# B&R Automation Studio project NAELD004C00R10L518F00 (part 37)

#### Act_Background.st
```iecst
(** 2019-01-21 **)
ACTION Act_Background:

	//Digital Input Mapping With Physical Input
	IF p_tyDISettings.diSafetyRlySig > 0 AND p_tyDISettings.diSafetyRlySig <= UDINT_TO_DINT(p_udiMax) THEN
		tyDInput.bSafetyRlySig	:= a_bPhysicalDI[p_tyDISettings.diSafetyRlySig];
	ELSE
		tyDInput.bSafetyRlySig	:= TRUE;
	END_IF

	IF p_tyDISettings.diEStopSig > 0 AND p_tyDISettings.diEStopSig <= UDINT_TO_DINT(p_udiMax) THEN
		tyDInput.bEStopSig	:= a_bPhysicalDI[p_tyDISettings.diEStopSig];
	ELSE
		tyDInput.bEStopSig	:= TRUE;
	END_IF

	IF p_tyDISettings.diCoverSWSig > 0 AND p_tyDISettings.diCoverSWSig <= UDINT_TO_DINT(p_udiMax) THEN
		tyDInput.bCoverSWSig	:= a_bPhysicalDI[p_tyDISettings.diCoverSWSig];
	ELSE
		tyDInput.bCoverSWSig	:= TRUE;
	END_IF

	IF bSelfTest = FALSE THEN
		IF p_tyDISettings.diDSBA > 0 AND p_tyDISettings.diDSBA <= UDINT_TO_DINT(p_udiMax) THEN
			tyDInput.bDSBA	:= a_bPhysicalDI[p_tyDISettings.diDSBA];
		ELSE
			tyDInput.bDSBA	:= FALSE;
		END_IF
	ELSE
		tyDInput.bDSBA	:= p_bPullConvHvBrd;
	END_IF

	IF p_tyDISettings.diDSBB > 0 AND p_tyDISettings.diDSBB <= UDINT_TO_DINT(p_udiMax) THEN
		tyDInput.bDSBB	:= a_bPhysicalDI[p_tyDISettings.diDSBB];
	ELSE
		tyDInput.bDSBB	:= FALSE;
	END_IF

	IF p_tyDISettings.diPullerExtRS > 0 AND p_tyDISettings.diPullerExtRS <= UDINT_TO_DINT(p_udiMax) THEN
		tyDInput.bPullerExtRS	:= a_bPhysicalDI[p_tyDISettings.diPullerExtRS];
	ELSE
		tyDInput.bPullerExtRS	:= FALSE;
	END_IF

	IF p_tyDISettings.diPullerRetRS > 0 AND p_tyDISettings.diPullerRetRS <= UDINT_TO_DINT(p_udiMax) THEN
		tyDInput.bPullerRetRS	:= a_bPhysicalDI[p_tyDISettings.diPullerRetRS];
	ELSE
		tyDInput.bPullerRetRS	:= TRUE;
	END_IF

	IF p_tyDISettings.diPullerRotHmRS > 0 AND p_tyDISettings.diPullerRotHmRS <= UDINT_TO_DINT(p_udiMax) THEN
		tyDInput.bPullerRotHmRS	:= a_bPhysicalDI[p_tyDISettings.diPullerRotHmRS];
	ELSE
		tyDInput.bPullerRotHmRS	:= TRUE;
	END_IF

	IF p_tyDISettings.diPullerRotRmRS > 0 AND p_tyDISettings.diPullerRotRmRS <= UDINT_TO_DINT(p_udiMax) THEN
		tyDInput.bPullerRotRmRS	:= a_bPhysicalDI[p_tyDISettings.diPullerRotRmRS];
	ELSE
		tyDInput.bPullerRotRmRS	:= FALSE;
	END_IF

	IF bSelfTest = FALSE THEN
		IF p_tyDISettings.diConvLftSen > 0 AND p_tyDISettings.diConvLftSen <= UDINT_TO_DINT(p_udiMax) THEN
			//Digital Input Filter
			fbConvLftSigFltr.tSigOnFltrTm	:= DINT_TO_TIME(p_diConvLftSenOnTm);
			fbConvLftSigFltr.tSigOffFltrTm	:= DINT_TO_TIME(p_diConvLftSenOffTm);
			fbConvLftSigFltr(bSigIn := a_bPhysicalDI[p_tyDISettings.diConvLftSen]);

			tyDInput.bConvLftSen	:= fbConvLftSigFltr.bSigOut;
		ELSE
			tyDInput.bConvLftSen	:= FALSE;
		END_IF
	ELSE
//		fbConvLftSenTm(IN:= p_bPullConvHvBrd);
//		IF EDGEPOS(p_bPullConvHvBrd) THEN
//			tyDInput.bConvLftSen	:= TRUE;
//		ELSIF fbConvLftSenTm.Q THEN
//			tyDInput.bConvLftSen	:= FALSE;
//		END_IF
	END_IF

	IF bSelfTest = FALSE THEN
		IF p_tyDISettings.diConvRgtSen > 0 AND p_tyDISettings.diConvRgtSen <= UDINT_TO_DINT(p_udiMax) THEN
			//Digital Input Filter
			fbConvRgtSigFltr.tSigOnFltrTm	:= DINT_TO_TIME(p_diConvRgtSenOnTm);
			fbConvRgtSigFltr.tSigOffFltrTm	:= DINT_TO_TIME(p_diConvRgtSenOffTm);
			fbConvRgtSigFltr(bSigIn := a_bPhysicalDI[p_tyDISettings.diConvRgtSen]);
			tyDInput.bConvRgtSen	:= fbConvRgtSigFltr.bSigOut;
		ELSE
			tyDInput.bConvRgtSen	:= FALSE;
		END_IF
	ELSE
		tyDInput.bConvRgtSen	:= p_bPullConvHvBrd;
	END_IF

	IF p_tyDISettings.diLifterTimingBeltSen > 0 AND p_tyDISettings.diLifterTimingBeltSen <= UDINT_TO_DINT(p_udiMax) THEN
		tyDInput.bLifterTimingBeltSen	:= a_bPhysicalDI[p_tyDISettings.diLifterTimingBeltSen];
	ELSE
		tyDInput.bLifterTimingBeltSen	:= TRUE;
	END_IF

	IF p_tyDISettings.diLifterSafetyLmtSW1 > 0 AND p_tyDISettings.diLifterSafetyLmtSW1 <= UDINT_TO_DINT(p_udiMax) THEN
		tyDInput.bLifterSafetyLmtSW1	:= a_bPhysicalDI[p_tyDISettings.diLifterSafetyLmtSW1];
	ELSE
		tyDInput.bLifterSafetyLmtSW1	:= TRUE;
	END_IF

	IF p_tyDISettings.diLifterSafetyLmtSW2 > 0 AND p_tyDISettings.diLifterSafetyLmtSW2 <= UDINT_TO_DINT(p_udiMax) THEN
		tyDInput.bLifterSafetyLmtSW2	:= a_bPhysicalDI[p_tyDISettings.diLifterSafetyLmtSW2];
	ELSE
		tyDInput.bLifterSafetyLmtSW2	:= TRUE;
	END_IF

	//Magazine 1 Fixed Clamper RSs
	IF p_tyDISettings.diMag1FixedClampRS > 0 AND p_tyDISettings.diMag1FixedClampRS <= UDINT_TO_DINT(p_udiMax) THEN
		tyDInput.bMag1FixedClampRS	:= a_bPhysicalDI[p_tyDISettings.diMag1FixedClampRS];
	ELSE
		tyDInput.bMag1FixedClampRS	:= FALSE;
	END_IF

	IF p_tyDISettings.diMag1FixedUnclampRS > 0 AND p_tyDISettings.diMag1FixedUnclampRS <= UDINT_TO_DINT(p_udiMax) THEN
		tyDInput.bMag1FixedUnclampRS	:= a_bPhysicalDI[p_tyDISettings.diMag1FixedUnclampRS];
	ELSE
		tyDInput.bMag1FixedUnclampRS	:= TRUE;
	END_IF

	//Magazine 1 Remote Clamper RSs
	IF p_tyDISettings.diMag1RemoteClampRS > 0 AND p_tyDISettings.diMag1RemoteClampRS <= UDINT_TO_DINT(p_udiMax) THEN
		tyDInput.bMag1RemoteClampRS	:= a_bPhysicalDI[p_tyDISettings.diMag1RemoteClampRS];
	ELSE
		tyDInput.bMag1RemoteClampRS	:= FALSE;
	END_IF

	IF p_tyDISettings.diMag1RemoteUnclampRS > 0 AND p_tyDISettings.diMag1RemoteUnclampRS <= UDINT_TO_DINT(p_udiMax) THEN
		tyDInput.bMag1RemoteUnclampRS	:= a_bPhysicalDI[p_tyDISettings.diMag1RemoteUnclampRS];
	ELSE
		tyDInput.bMag1RemoteUnclampRS	:= TRUE;
	END_IF

	//Magazine 1 Sel Clamper RSs
	IF p_tyDISettings.diMag1SelUnClampRS > 0 AND p_tyDISettings.diMag1SelUnClampRS <= UDINT_TO_DINT(p_udiMax) THEN
		tyDInput.bMag1SelUnClampRS	:= a_bPhysicalDI[p_tyDISettings.diMag1SelUnClampRS];
	ELSE
		tyDInput.bMag1SelUnClampRS	:= FALSE;
	END_IF

	//Magazine 2 Fixed Clamper RSs
	IF p_tyDISettings.diMag2FixedClampRS > 0 AND p_tyDISettings.diMag2FixedClampRS <= UDINT_TO_DINT(p_udiMax) THEN
		tyDInput.bMag2FixedClampRS	:= a_bPhysicalDI[p_tyDISettings.diMag2FixedClampRS];
	ELSE
		tyDInput.bMag2FixedClampRS	:= FALSE;
	END_IF

	IF p_tyDISettings.diMag2FixedUnclampRS > 0 AND p_tyDISettings.diMag2FixedUnclampRS <= UDINT_TO_DINT(p_udiMax) THEN
		tyDInput.bMag2FixedUnclampRS	:= a_bPhysicalDI[p_tyDISettings.diMag2FixedUnclampRS];
	ELSE
		tyDInput.bMag2FixedUnclampRS	:= TRUE;
	END_IF

	//Magazine 2 Remote Clamper RSs
	IF p_tyDISettings.diMag2RemoteClampRS > 0 AND p_tyDISettings.diMag2RemoteClampRS <= UDINT_TO_DINT(p_udiMax) THEN
		tyDInput.bMag2RemoteClampRS	:= a_bPhysicalDI[p_tyDISettings.diMag2RemoteClampRS];
	ELSE
		tyDInput.bMag2RemoteClampRS	:= FALSE;
	END_IF

	IF p_tyDISettings.diMag2RemoteUnclampRS > 0 AND p_tyDISettings.diMag2RemoteUnclampRS <= UDINT_TO_DINT(p_udiMax) THEN
		tyDInput.bMag2RemoteUnclampRS	:= a_bPhysicalDI[p_tyDISettings.diMag2RemoteUnclampRS];
	ELSE
		tyDInput.bMag2RemoteUnclampRS	:= TRUE;
	END_IF

	//Magazine 2 Sel Clamper RSs
	IF p_tyDISettings.diMag2SelUnClampRS > 0 AND p_tyDISettings.diMag2SelUnClampRS <= UDINT_TO_DINT(p_udiMax) THEN
		tyDInput.bMag2SelUnClampRS	:= a_bPhysicalDI[p_tyDISettings.diMag2SelUnClampRS];
	ELSE
		tyDInput.bMag2SelUnClampRS	:= FALSE;
	END_IF

	//Magazine 3 Fixed Clamper RSs
	IF p_tyDISettings.diMag3FixedClampRS > 0 AND p_tyDISettings.diMag3FixedClampRS <= UDINT_TO_DINT(p_udiMax) THEN
		tyDInput.bMag3FixedClampRS	:= a_bPhysicalDI[p_tyDISettings.diMag3FixedClampRS];
	ELSE
		tyDInput.bMag3FixedClampRS	:= FALSE;
	END_IF

	IF p_tyDISettings.diMag3FixedUnclampRS > 0 AND p_tyDISettings.diMag3FixedUnclampRS <= UDINT_TO_DINT(p_udiMax) THEN
		tyDInput.bMag3FixedUnclampRS	:= a_bPhysicalDI[p_tyDISettings.diMag3FixedUnclampRS];
	ELSE
		tyDInput.bMag3FixedUnclampRS	:= TRUE;
	END_IF

	//Magazine 3 Remote Clamper RSs
	IF p_tyDISettings.diMag3RemoteClampRS > 0 AND p_tyDISettings.diMag3RemoteClampRS <= UDINT_TO_DINT(p_udiMax) THEN
		tyDInput.bMag3RemoteClampRS	:= a_bPhysicalDI[p_tyDISettings.diMag3RemoteClampRS];
	ELSE
		tyDInput.bMag3RemoteClampRS	:= FALSE;
	END_IF

	IF p_tyDISettings.diMag3RemoteUnclampRS > 0 AND p_tyDISettings.diMag3RemoteUnclampRS <= UDINT_TO_DINT(p_udiMax) THEN
		tyDInput.bMag3RemoteUnclampRS	:= a_bPhysicalDI[p_tyDISettings.diMag3RemoteUnclampRS];
	ELSE
		tyDInput.bMag3RemoteUnclampRS	:= TRUE;
	END_IF

	//Magazine 3 Sel Clamper RSs
	IF p_tyDISettings.diMag3SelUnClampRS > 0 AND p_tyDISettings.diMag3SelUnClampRS <= UDINT_TO_DINT(p_udiMax) THEN
		tyDInput.bMag3SelUnClampRS	:= a_bPhysicalDI[p_tyDISettings.diMag3SelUnClampRS];
	ELSE
		tyDInput.bMag3SelUnClampRS	:= FALSE;
	END_IF

	//Magazine 4 Fixed Clamper RSs
	IF p_tyDISettings.diMag4FixedClampRS > 0 AND p_tyDISettings.diMag4FixedClampRS <= UDINT_TO_DINT(p_udiMax) THEN
		tyDInput.bMag4FixedClampRS	:= a_bPhysicalDI[p_tyDISettings.diMag4FixedClampRS];
	ELSE
		tyDInput.bMag4FixedClampRS	:= FALSE;
	END_IF

	IF p_tyDISettings.diMag4FixedUnclampRS > 0 AND p_tyDISettings.diMag4FixedUnclampRS <= UDINT_TO_DINT(p_udiMax) THEN
		tyDInput.bMag4FixedUnclampRS	:= a_bPhysicalDI[p_tyDISettings.diMag4FixedUnclampRS];
	ELSE
		tyDInput.bMag4FixedUnclampRS	:= TRUE;
	END_IF

	//Magazine 4 Remote Clamper RSs
	IF p_tyDISettings.diMag4RemoteClampRS > 0 AND p_tyDISettings.diMag4RemoteClampRS <= UDINT_TO_DINT(p_udiMax) THEN
		tyDInput.bMag4RemoteClampRS	:= a_bPhysicalDI[p_tyDISettings.diMag4RemoteClampRS];
	ELSE
		tyDInput.bMag4RemoteClampRS	:= FALSE;
	END_IF

	IF p_tyDISettings.diMag4RemoteUnclampRS > 0 AND p_tyDISettings.diMag4RemoteUnclampRS <= UDINT_TO_DINT(p_udiMax) THEN
		tyDInput.bMag4RemoteUnclampRS	:= a_bPhysicalDI[p_tyDISettings.diMag4RemoteUnclampRS];
	ELSE
		tyDInput.bMag4RemoteUnclampRS	:= TRUE;
	END_IF

	//Magazine 4 Sel Clamper RSs
	IF p_tyDISettings.diMag4SelUnClampRS > 0 AND p_tyDISettings.diMag4SelUnClampRS <= UDINT_TO_DINT(p_udiMax) THEN
		tyDInput.bMag4SelUnClampRS	:= a_bPhysicalDI[p_tyDISettings.diMag4SelUnClampRS];
	ELSE
		tyDInput.bMag4SelUnClampRS	:= FALSE;
	END_IF

	IF p_tyDISettings.diInShutterOpenRS > 0 AND p_tyDISettings.diInShutterOpenRS <= UDINT_TO_DINT(p_udiMax) THEN
		tyDInput.bInShutterOpenRS	:= a_bPhysicalDI[p_tyDISettings.diInShutterOpenRS];
	ELSE
		tyDInput.bInShutterOpenRS	:= FALSE;
	END_IF

	IF p_tyDISettings.diInShutterCloseRS > 0 AND p_tyDISettings.diInShutterCloseRS <= UDINT_TO_DINT(p_udiMax) THEN
		tyDInput.bInShutterCloseRS	:= a_bPhysicalDI[p_tyDISettings.diInShutterCloseRS];
	ELSE
		tyDInput.bInShutterCloseRS	:= FALSE;
	END_IF

	IF p_tyDISettings.diOutShutterOpenRS > 0 AND p_tyDISettings.diOutShutterOpenRS <= UDINT_TO_DINT(p_udiMax) THEN
		tyDInput.bOutShutterOpenRS	:= a_bPhysicalDI[p_tyDISettings.diOutShutterOpenRS];
	ELSE
		tyDInput.bOutShutterOpenRS	:= FALSE;
	END_IF

	IF p_tyDISettings.diOutShutterCloseRS > 0 AND p_tyDISettings.diOutShutterCloseRS <= UDINT_TO_DINT(p_udiMax) THEN
		tyDInput.bOutShutterCloseRS	:= a_bPhysicalDI[p_tyDISettings.diOutShutterCloseRS];
	ELSE
		tyDInput.bOutShutterCloseRS	:= FALSE;
	END_IF

	IF bSelfTest = FALSE THEN
		IF p_tyDISettings.diMagPresentSen1 > 0 AND p_tyDISettings.diMagPresentSen1 <= UDINT_TO_DINT(p_udiMax) THEN
			//Digital Input Filter
			fbMagConv1PresentSigFltr.tSigOnFltrTm	:= DINT_TO_TIME(p_diMagConvPresentSenOnTm);
			fbMagConv1PresentSigFltr.tSigOffFltrTm	:= DINT_TO_TIME(p_diMagConvPresentSenOffTm);
			fbMagConv1PresentSigFltr(bSigIn := a_bPhysicalDI[p_tyDISettings.diMagPresentSen1]);
			tyDInput.bMagPresentSen1	:= fbMagConv1PresentSigFltr.bSigOut;
		//	tyDInput.bMagPresentSen1	:= a_bPhysicalDI[p_tyDISettings.diMagPresentSen1];
		ELSE
			tyDInput.bMagPresentSen1	:= FALSE;
		END_IF

		IF p_tyDISettings.diMagPresentSen2 > 0 AND p_tyDISettings.diMagPresentSen2 <= UDINT_TO_DINT(p_udiMax) THEN
			fbMagConv2PresentSigFltr.tSigOnFltrTm	:= DINT_TO_TIME(p_diMagConvPresentSenOnTm);
			fbMagConv2PresentSigFltr.tSigOffFltrTm	:= DINT_TO_TIME(p_diMagConvPresentSenOffTm);
			fbMagConv2PresentSigFltr(bSigIn := a_bPhysicalDI[p_tyDISettings.diMagPresentSen2]);
			tyDInput.bMagPresentSen2	:= fbMagConv2PresentSigFltr.bSigOut;
			//	tyDInput.bMagPresentSen2	:= a_bPhysicalDI[p_tyDISettings.diMagPresentSen2];
		ELSE
			tyDInput.bMagPresentSen2	:= FALSE;
		END_IF

		IF p_tyDISettings.diMagPresentSen3 > 0 AND p_tyDISettings.diMagPresentSen3 <= UDINT_TO_DINT(p_udiMax) THEN
			fbMagConv3PresentSigFltr.tSigOnFltrTm	:= DINT_TO_TIME(p_diMagConvPresentSenOnTm);
			fbMagConv3PresentSigFltr.tSigOffFltrTm	:= DINT_TO_TIME(p_diMagConvPresentSenOffTm);
			fbMagConv3PresentSigFltr(bSigIn := a_bPhysicalDI[p_tyDISettings.diMagPresentSen3]);
			tyDInput.bMagPresentSen3	:= fbMagConv3PresentSigFltr.bSigOut;
			//	tyDInput.bMagPresentSen3	:= a_bPhysicalDI[p_tyDISettings.diMagPresentSen3];
		ELSE
			tyDInput.bMagPresentSen3	:= FALSE;
		END_IF

		IF p_tyDISettings.diMagPresentSen4 > 0 AND p_tyDISettings.diMagPresentSen4 <= UDINT_TO_DINT(p_udiMax) THEN
			//Digital Input Filter
			fbMagConv4PresentSigFltr.tSigOnFltrTm	:= DINT_TO_TIME(p_diMagConvPresentSenOnTm);
			fbMagConv4PresentSigFltr.tSigOffFltrTm	:= DINT_TO_TIME(p_diMagConvPresentSenOffTm);
			fbMagConv4PresentSigFltr(bSigIn := a_bPhysicalDI[p_tyDISettings.diMagPresentSen4]);
			tyDInput.bMagPresentSen4	:= fbMagConv4PresentSigFltr.bSigOut;
			//	tyDInput.bMagPresentSen4	:= a_bPhysicalDI[p_tyDISettings.diMagPresentSen4];
		ELSE
			tyDInput.bMagPresentSen4	:= FALSE;
		END_IF

		IF p_tyDISettings.diMagConvEntSen1 > 0 AND p_tyDISettings.diMagConvEntSen1 <= UDINT_TO_DINT(p_udiMax) THEN
			//Digital Input Filter
			fbMagConv1EntSigFltr.tSigOnFltrTm	:= DINT_TO_TIME(p_diMagConvEntSenOnTm);
			fbMagConv1EntSigFltr.tSigOffFltrTm	:= DINT_TO_TIME(p_diMagConvEntSenOffTm);
			fbMagConv1EntSigFltr(bSigIn := a_bPhysicalDI[p_tyDISettings.diMagConvEntSen1]);
			tyDInput.bMagConvEntSen1	:= fbMagConv1EntSigFltr.bSigOut;
		ELSE
			tyDInput.bMagConvEntSen1	:= FALSE;
		END_IF

		IF p_tyDISettings.diMagConvEntSen2 > 0 AND p_tyDISettings.diMagConvEntSen2 <= UDINT_TO_DINT(p_udiMax) THEN
			//Digital Input Filter
			fbMagConv2EntSigFltr.tSigOnFltrTm	:= DINT_TO_TIME(p_diMagConvEntSenOnTm);
			fbMagConv2EntSigFltr.tSigOffFltrTm	:= DINT_TO_TIME(p_diMagConvEntSenOffTm);
			fbMagConv2EntSigFltr(bSigIn := a_bPhysicalDI[p_tyDISettings.diMagConvEntSen2]);
			tyDInput.bMagConvEntSen2	:= fbMagConv2EntSigFltr.bSigOut;
		ELSE
			tyDInput.bMagConvEntSen2	:= FALSE;
		END_IF

		IF p_tyDISettings.diMagConvEntSen3 > 0 AND p_tyDISettings.diMagConvEntSen3 <= UDINT_TO_DINT(p_udiMax) THEN
			//Digital Input Filter
			fbMagConv3EntSigFltr.tSigOnFltrTm	:= DINT_TO_TIME(p_diMagConvEntSenOnTm);
			fbMagConv3EntSigFltr.tSigOffFltrTm	:= DINT_TO_TIME(p_diMagConvEntSenOffTm);
			fbMagConv3EntSigFltr(bSigIn := a_bPhysicalDI[p_tyDISettings.diMagConvEntSen3]);
			tyDInput.bMagConvEntSen3	:= fbMagConv3EntSigFltr.bSigOut;
		ELSE
			tyDInput.bMagConvEntSen3	:= FALSE;
		END_IF

		IF p_tyDISettings.diMagConvEntSen4 > 0 AND p_tyDISettings.diMagConvEntSen4 <= UDINT_TO_DINT(p_udiMax) THEN
			//Digital Input Filter
			fbMagConv4EntSigFltr.tSigOnFltrTm	:= DINT_TO_TIME(p_diMagConvEntSenOnTm);
			fbMagConv4EntSigFltr.tSigOffFltrTm	:= DINT_TO_TIME(p_diMagConvEntSenOffTm);
			fbMagConv4EntSigFltr(bSigIn := a_bPhysicalDI[p_tyDISettings.diMagConvEntSen4]);
			tyDInput.bMagConvEntSen4	:= fbMagConv4EntSigFltr.bSigOut;
		ELSE
			tyDInput.bMagConvEntSen4	:= FALSE;
		END_IF

	ELSE

		CASE p_eLDMag OF
			LDMagDual:

				fbSelfTestTm1(IN:= p_tyDO.bMag1ConvMtrIn = FALSE  AND p_tyDO.bMag1ConvMtrOut = FALSE);
				IF fbSelfTestTm1.Q THEN
					tyDInput.bMagPresentSen1 := TRUE;
				ELSIF p_tyDO.bMag1ConvMtrOut THEN
					tyDInput.bMagPresentSen1 := FALSE;
					tyDInput.bMagConvEntSen1 := TRUE;
				ELSIF tyDInput.bMagConvEntSen1 THEN
					tyDInput.bMagConvEntSen1 := FALSE;
				END_IF

				fbSelfTestTm2(IN:= p_tyDO.bMag2ConvMtrIn = FALSE  AND p_tyDO.bMag2ConvMtrOut = FALSE);
				IF fbSelfTestTm2.Q THEN
					tyDInput.bMagPresentSen2 := TRUE;
				ELSIF p_tyDO.bMag2ConvMtrOut THEN
					tyDInput.bMagPresentSen2 := FALSE;
					tyDInput.bMagConvEntSen2 := TRUE;
				ELSIF tyDInput.bMagConvEntSen2 THEN
					tyDInput.bMagConvEntSen2 := FALSE;
				END_IF

			LDMagTriple:

				fbSelfTestTm1(IN:= p_tyDO.bMag1ConvMtrIn = FALSE  AND p_tyDO.bMag1ConvMtrOut = FALSE);
				IF fbSelfTestTm1.Q THEN
					tyDInput.bMagPresentSen1 := TRUE;
				ELSIF p_tyDO.bMag1ConvMtrOut THEN
					tyDInput.bMagPresentSen1 := FALSE;
					tyDInput.bMagConvEntSen1 := TRUE;
				ELSIF tyDInput.bMagConvEntSen1 THEN
					tyDInput.bMagConvEntSen1 := FALSE;
				END_IF

				fbSelfTestTm2(IN:= p_tyDO.bMag2ConvMtrIn = FALSE  AND p_tyDO.bMag2ConvMtrOut = FALSE);
				IF fbSelfTestTm2.Q THEN
					tyDInput.bMagPresentSen2 := TRUE;
				ELSIF p_tyDO.bMag2ConvMtrOut THEN
					tyDInput.bMagPresentSen2 := FALSE;
					tyDInput.bMagConvEntSen2 := TRUE;
				ELSIF tyDInput.bMagConvEntSen2 THEN
					tyDInput.bMagConvEntSen2 := FALSE;
				END_IF

				fbSelfTestTm3(IN:= p_tyDO.bMag3ConvMtrIn = FALSE  AND p_tyDO.bMag3ConvMtrOut = FALSE);
				IF fbSelfTestTm3.Q THEN
					tyDInput.bMagPresentSen3 := TRUE;
				ELSIF p_tyDO.bMag3ConvMtrOut THEN
					tyDInput.bMagPresentSen3 := FALSE;
					tyDInput.bMagConvEntSen3 := TRUE;
				ELSIF tyDInput.bMagConvEntSen3 THEN
					tyDInput.bMagConvEntSen3 := FALSE;
				END_IF

			LDMagQuadruple:

				fbSelfTestTm1(IN:= p_tyDO.bMag1ConvMtrIn = FALSE  AND p_tyDO.bMag1ConvMtrOut = FALSE);
				IF fbSelfTestTm1.Q THEN
					tyDInput.bMagPresentSen1 := TRUE;
				ELSIF p_tyDO.bMag1ConvMtrOut THEN
					tyDInput.bMagPresentSen1 := FALSE;
					tyDInput.bMagConvEntSen1 := TRUE;
				ELSIF tyDInput.bMagConvEntSen1 THEN
					tyDInput.bMagConvEntSen1 := FALSE;
				END_IF

				fbSelfTestTm2(IN:= p_tyDO.bMag2ConvMtrIn = FALSE  AND p_tyDO.bMag2ConvMtrOut = FALSE);
				IF fbSelfTestTm2.Q THEN
					tyDInput.bMagPresentSen2 := TRUE;
				ELSIF p_tyDO.bMag2ConvMtrOut THEN
					tyDInput.bMagPresentSen2 := FALSE;
					tyDInput.bMagConvEntSen2 := TRUE;
				ELSIF tyDInput.bMagConvEntSen2 THEN
					tyDInput.bMagConvEntSen2 := FALSE;
				END_IF

				fbSelfTestTm3(IN:= p_tyDO.bMag3ConvMtrIn = FALSE  AND p_tyDO.bMag3ConvMtrOut = FALSE);
				IF fbSelfTestTm3.Q THEN
					tyDInput.bMagPresentSen3 := TRUE;
				ELSIF p_tyDO.bMag3ConvMtrOut THEN
					tyDInput.bMagPresentSen3 := FALSE;
					tyDInput.bMagConvEntSen3 := TRUE;
				ELSIF tyDInput.bMagConvEntSen3 THEN
					tyDInput.bMagConvEntSen3 := FALSE;
				END_IF

				fbSelfTestTm4(IN:= p_tyDO.bMag4ConvMtrIn = FALSE  AND p_tyDO.bMag4ConvMtrOut = FALSE);
				IF fbSelfTestTm4.Q THEN
					tyDInput.bMagPresentSen4 := TRUE;
				ELSIF p_tyDO.bMag4ConvMtrOut THEN
					tyDInput.bMagPresentSen4 := FALSE;
					tyDInput.bMagConvEntSen4 := TRUE;
				ELSIF tyDInput.bMagConvEntSen4 THEN
					tyDInput.bMagConvEntSen4 := FALSE;
				END_IF
		END_CASE
	END_IF

	IF p_tyDISettings.diMag1AGVInPosSen1 > 0 AND p_tyDISettings.diMag1AGVInPosSen1 <= UDINT_TO_DINT(p_udiMax) THEN
		tyDInput.bMag1AGVInPosSen1	:= a_bPhysicalDI[p_tyDISettings.diMag1AGVInPosSen1];
	ELSE
		tyDInput.bMag1AGVInPosSen1	:= FALSE;
	END_IF

	IF p_tyDISettings.diMag1AGVInPosSen2 > 0 AND p_tyDISettings.diMag1AGVInPosSen2 <= UDINT_TO_DINT(p_udiMax) THEN
		tyDInput.bMag1AGVInPosSen2	:= a_bPhysicalDI[p_tyDISettings.diMag1AGVInPosSen2];
	ELSE
		tyDInput.bMag1AGVInPosSen2	:= FALSE;
	END_IF

	IF p_tyDISettings.diMag2AGVInPosSen1 > 0 AND p_tyDISettings.diMag2AGVInPosSen1 <= UDINT_TO_DINT(p_udiMax) THEN
		tyDInput.bMag2AGVInPosSen1	:= a_bPhysicalDI[p_tyDISettings.diMag2AGVInPosSen1];
	ELSE
		tyDInput.bMag2AGVInPosSen1	:= FALSE;
	END_IF

	IF p_tyDISettings.diMag2AGVInPosSen2 > 0 AND p_tyDISettings.diMag2AGVInPosSen2 <= UDINT_TO_DINT(p_udiMax) THEN
		tyDInput.bMag2AGVInPosSen2	:= a_bPhysicalDI[p_tyDISettings.diMag2AGVInPosSen2];
	ELSE
		tyDInput.bMag2AGVInPosSen2	:= FALSE;
	END_IF

	IF p_tyDISettings.diMag3AGVInPosSen1 > 0 AND p_tyDISettings.diMag3AGVInPosSen1 <= UDINT_TO_DINT(p_udiMax) THEN
		tyDInput.bMag3AGVInPosSen1	:= a_bPhysicalDI[p_tyDISettings.diMag3AGVInPosSen1];
	ELSE
		tyDInput.bMag3AGVInPosSen1	:= FALSE;
	END_IF

	IF p_tyDISettings.diMag3AGVInPosSen2 > 0 AND p_tyDISettings.diMag3AGVInPosSen2 <= UDINT_TO_DINT(p_udiMax) THEN
		tyDInput.bMag3AGVInPosSen2	:= a_bPhysicalDI[p_tyDISettings.diMag3AGVInPosSen2];
	ELSE
		tyDInput.bMag3AGVInPosSen2	:= FALSE;
	END_IF

	IF p_tyDISettings.diMag1OrientChkSen1 > 0 AND p_tyDISettings.diMag1OrientChkSen1 <= UDINT_TO_DINT(p_udiMax) THEN
		tyDInput.bMag1OrientChkSen1	:= a_bPhysicalDI[p_tyDISettings.diMag1OrientChkSen1];
	ELSE
		tyDInput.bMag1OrientChkSen1	:= FALSE;
	END_IF

	IF p_tyDISettings.diMag1OrientChkSen2 > 0 AND p_tyDISettings.diMag1OrientChkSen2 <= UDINT_TO_DINT(p_udiMax) THEN
		tyDInput.bMag1OrientChkSen2	:= a_bPhysicalDI[p_tyDISettings.diMag1OrientChkSen2];
	ELSE
		tyDInput.bMag1OrientChkSen2	:= FALSE;
	END_IF

	IF p_tyDISettings.diMag2OrientChkSen1 > 0 AND p_tyDISettings.diMag2OrientChkSen1 <= UDINT_TO_DINT(p_udiMax) THEN
		tyDInput.bMag2OrientChkSen1	:= a_bPhysicalDI[p_tyDISettings.diMag2OrientChkSen1];
	ELSE
		tyDInput.bMag2OrientChkSen1	:= FALSE;
	END_IF

	IF p_tyDISettings.diMag2OrientChkSen2 > 0 AND p_tyDISettings.diMag2OrientChkSen2 <= UDINT_TO_DINT(p_udiMax) THEN
		tyDInput.bMag2OrientChkSen2	:= a_bPhysicalDI[p_tyDISettings.diMag2OrientChkSen2];
	ELSE
		tyDInput.bMag2OrientChkSen2	:= FALSE;
	END_IF

	IF p_tyDISettings.diMag3OrientChkSen1 > 0 AND p_tyDISettings.diMag3OrientChkSen1 <= UDINT_TO_DINT(p_udiMax) THEN
		tyDInput.bMag3OrientChkSen1	:= a_bPhysicalDI[p_tyDISettings.diMag3OrientChkSen1];
	ELSE
		tyDInput.bMag3OrientChkSen1	:= FALSE;
	END_IF

	IF p_tyDISettings.diMag3OrientChkSen2 > 0 AND p_tyDISettings.diMag3OrientChkSen2 <= UDINT_TO_DINT(p_udiMax) THEN
		tyDInput.bMag3OrientChkSen2	:= a_bPhysicalDI[p_tyDISettings.diMag3OrientChkSen2];
	ELSE
		tyDInput.bMag3OrientChkSen2	:= FALSE;
	END_IF

	IF p_tyDISettings.diDSWidthChkSen > 0 AND p_tyDISettings.diDSWidthChkSen <= UDINT_TO_DINT(p_udiMax) THEN
		tyDInput.bDSWidthChkSen	:= a_bPhysicalDI[p_tyDISettings.diDSWidthChkSen];
	ELSE
		tyDInput.bDSWidthChkSen	:= FALSE;
	END_IF

	//Magazine 1 Height Sensor
	IF p_tyDISettings.diMagConvHeightSen1 > 0 AND p_tyDISettings.diMagConvHeightSen1 <= UDINT_TO_DINT(p_udiMax) THEN
		tyDInput.bMagConvHeightSen1	:= a_bPhysicalDI[p_tyDISettings.diMagConvHeightSen1];
	ELSE
		tyDInput.bMagConvHeightSen1	:= FALSE;
	END_IF

	//Magazine 2 Height Sensor
	IF p_tyDISettings.diMagConvHeightSen2 > 0 AND p_tyDISettings.diMagConvHeightSen2 <= UDINT_TO_DINT(p_udiMax) THEN
		tyDInput.bMagConvHeightSen2	:= a_bPhysicalDI[p_tyDISettings.diMagConvHeightSen2];
	ELSE
		tyDInput.bMagConvHeightSen2	:= FALSE;
	END_IF

	//Magazine 3 Height Sensor
	IF p_tyDISettings.diMagConvHeightSen3 > 0 AND p_tyDISettings.diMagConvHeightSen3 <= UDINT_TO_DINT(p_udiMax) THEN
		tyDInput.bMagConvHeightSen3	:= a_bPhysicalDI[p_tyDISettings.diMagConvHeightSen3];
	ELSE
		tyDInput.bMagConvHeightSen3	:= FALSE;
	END_IF

	//Magazine 4 Height Sensor
	IF p_tyDISettings.diMagConvHeightSen4 > 0 AND p_tyDISettings.diMagConvHeightSen4 <= UDINT_TO_DINT(p_udiMax) THEN
		tyDInput.bMagConvHeightSen4	:= a_bPhysicalDI[p_tyDISettings.diMagConvHeightSen4];
	ELSE
		tyDInput.bMagConvHeightSen4	:= FALSE;
	END_IF

	//Magazine 1 Small Sensor
	IF p_tyDISettings.diMagConvSmallMagSen1 > 0 AND p_tyDISettings.diMagConvSmallMagSen1 <= UDINT_TO_DINT(p_udiMax) THEN
		tyDInput.bMagConvSmallMagSen1	:= a_bPhysicalDI[p_tyDISettings.diMagConvSmallMagSen1];
	ELSE
		tyDInput.bMagConvSmallMagSen1	:= FALSE;
	END_IF

	//Magazine 2 Small Sensor
	IF p_tyDISettings.diMagConvSmallMagSen2 > 0 AND p_tyDISettings.diMagConvSmallMagSen2 <= UDINT_TO_DINT(p_udiMax) THEN
		tyDInput.bMagConvSmallMagSen2	:= a_bPhysicalDI[p_tyDISettings.diMagConvSmallMagSen2];
	ELSE
		tyDInput.bMagConvSmallMagSen2	:= FALSE;
	END_IF

	//Magazine 3 Small Sensor
	IF p_tyDISettings.diMagConvSmallMagSen3 > 0 AND p_tyDISettings.diMagConvSmallMagSen3 <= UDINT_TO_DINT(p_udiMax) THEN
		tyDInput.bMagConvSmallMagSen3	:= a_bPhysicalDI[p_tyDISettings.diMagConvSmallMagSen3];
	ELSE
		tyDInput.bMagConvSmallMagSen3	:= FALSE;
	END_IF

	//Magazine 4 Small Sensor
	IF p_tyDISettings.diMagConvSmallMagSen4 > 0 AND p_tyDISettings.diMagConvSmallMagSen4 <= UDINT_TO_DINT(p_udiMax) THEN
		tyDInput.bMagConvSmallMagSen4	:= a_bPhysicalDI[p_tyDISettings.diMagConvSmallMagSen4];
	ELSE
		tyDInput.bMagConvSmallMagSen4	:= FALSE;
	END_IF

	//Magazine 1 Large Sensor
	IF p_tyDISettings.diMagConvLargeMagSen1 > 0 AND p_tyDISettings.diMagConvLargeMagSen1 <= UDINT_TO_DINT(p_udiMax) THEN
		tyDInput.bMagConvLargeMagSen1	:= a_bPhysicalDI[p_tyDISettings.diMagConvLargeMagSen1];
	ELSE
		tyDInput.bMagConvLargeMagSen1	:= FALSE;
	END_IF

	//Magazine 2 Large Sensor
	IF p_tyDISettings.diMagConvLargeMagSen2 > 0 AND p_tyDISettings.diMagConvLargeMagSen2 <= UDINT_TO_DINT(p_udiMax) THEN
		tyDInput.bMagConvLargeMagSen2	:= a_bPhysicalDI[p_tyDISettings.diMagConvLargeMagSen2];
	ELSE
		tyDInput.bMagConvLargeMagSen2	:= FALSE;
	END_IF

	//Magazine 3 Large Sensor
	IF p_tyDISettings.diMagConvLargeMagSen3 > 0 AND p_tyDISettings.diMagConvLargeMagSen3 <= UDINT_TO_DINT(p_udiMax) THEN
		tyDInput.bMagConvLargeMagSen3	:= a_bPhysicalDI[p_tyDISettings.diMagConvLargeMagSen3];
	ELSE
		tyDInput.bMagConvLargeMagSen3	:= FALSE;
	END_IF

	//Magazine 4 Large Sensor
	IF p_tyDISettings.diMagConvLargeMagSen4 > 0 AND p_tyDISettings.diMagConvLargeMagSen4 <= UDINT_TO_DINT(p_udiMax) THEN
		tyDInput.bMagConvLargeMagSen4	:= a_bPhysicalDI[p_tyDISettings.diMagConvLargeMagSen4];
	ELSE
		tyDInput.bMagConvLargeMagSen4	:= FALSE;
	END_IF

	//Magazine 1 CAB717.2 Sensor
	IF p_tyDISettings.diMagConvCAB717MagSen1 > 0 AND p_tyDISettings.diMagConvCAB717MagSen1 <= UDINT_TO_DINT(p_udiMax) THEN
		tyDInput.bMagConvCAB717MagSen1	:= a_bPhysicalDI[p_tyDISettings.diMagConvCAB717MagSen1];
	ELSE
		tyDInput.bMagConvCAB717MagSen1	:= FALSE;
	END_IF

	//Magazine 2 CAB717.2 Sensor
	IF p_tyDISettings.diMagConvCAB717MagSen2 > 0 AND p_tyDISettings.diMagConvCAB717MagSen2 <= UDINT_TO_DINT(p_udiMax) THEN
		tyDInput.bMagConvCAB717MagSen2	:= a_bPhysicalDI[p_tyDISettings.diMagConvCAB717MagSen2];
	ELSE
		tyDInput.bMagConvCAB717MagSen2	:= FALSE;
	END_IF

	//Magazine 3 CAB717.2 Sensor
	IF p_tyDISettings.diMagConvCAB717MagSen3 > 0 AND p_tyDISettings.diMagConvCAB717MagSen3 <= UDINT_TO_DINT(p_udiMax) THEN
		tyDInput.bMagConvCAB717MagSen3	:= a_bPhysicalDI[p_tyDISettings.diMagConvCAB717MagSen3];
	ELSE
		tyDInput.bMagConvCAB717MagSen3	:= FALSE;
	END_IF

	//Magazine 4 CAB717.2 Sensor
	IF p_tyDISettings.diMagConvCAB717MagSen4 > 0 AND p_tyDISettings.diMagConvCAB717MagSen4 <= UDINT_TO_DINT(p_udiMax) THEN
		tyDInput.bMagConvCAB717MagSen4	:= a_bPhysicalDI[p_tyDISettings.diMagConvCAB717MagSen4];
	ELSE
		tyDInput.bMagConvCAB717MagSen4	:= FALSE;
	END_IF

	CASE p_eLinkAGVComProtocol OF
		McSetAGVCommOPCUA:
			tyDInput.bFleetManagerReady	:= p_tyTagFromMes.bActive;

		McSetAGVCommHardIO:
			//Fleet Manager Active Status
			IF p_tyDISettings.diFleetManagerReady > 0 AND p_tyDISettings.diFleetManagerReady <= UDINT_TO_DINT(p_udiMax) THEN
				tyDInput.bFleetManagerReady	:= a_bPhysicalDI[p_tyDISettings.diFleetManagerReady];
			ELSE
				tyDInput.bFleetManagerReady	:= FALSE;
			END_IF

		McSetAGVCommDisabled:
			tyDInput.bFleetManagerReady	:= FALSE;
	END_CASE

	IF p_bLinkNtParamProjSOTSenPrep OR p_eLinkAGVComProtocol = McSetAGVCommHardIO THEN
			IF p_bUIAGVSimulationOn = FALSE THEN
				//SOT Configuration
				IF p_tyDISettings.diSOT1Receive > 0 AND p_tyDISettings.diSOT1Receive <= UDINT_TO_DINT(p_udiMax) THEN
					tyDInput.bSOT1Receive	:= a_bPhysicalDI[p_tyDISettings.diSOT1Receive];
				ELSE
					tyDInput.bSOT1Receive	:= FALSE;
				END_IF

				IF p_tyDISettings.diSOT1AIVError > 0 AND p_tyDISettings.diSOT1AIVError <= UDINT_TO_DINT(p_udiMax) THEN
					tyDInput.bSOT1AIVError	:= a_bPhysicalDI[p_tyDISettings.diSOT1AIVError];
				ELSE
					tyDInput.bSOT1AIVError	:= FALSE;
				END_IF

				IF p_tyDISettings.diSOT1AIVSizeLarge > 0 AND p_tyDISettings.diSOT1AIVSizeLarge <= UDINT_TO_DINT(p_udiMax) THEN
					tyDInput.bSOT1AIVSizeLarge	:= a_bPhysicalDI[p_tyDISettings.diSOT1AIVSizeLarge];
				ELSE
					tyDInput.bSOT1AIVSizeLarge	:= FALSE;
				END_IF

				IF p_tyDISettings.diSOT1AIVReady > 0 AND p_tyDISettings.diSOT1AIVReady <= UDINT_TO_DINT(p_udiMax) THEN
					tyDInput.bSOT1AIVReady	:= a_bPhysicalDI[p_tyDISettings.diSOT1AIVReady];
				ELSE
					tyDInput.bSOT1AIVReady	:= FALSE;
				END_IF

				IF p_tyDISettings.diSOT1AIVAvailable > 0 AND p_tyDISettings.diSOT1AIVAvailable <= UDINT_TO_DINT(p_udiMax) THEN
					tyDInput.bSOT1AIVAvailable	:= a_bPhysicalDI[p_tyDISettings.diSOT1AIVAvailable];
				ELSE
					tyDInput.bSOT1AIVAvailable	:= FALSE;
				END_IF

				IF p_tyDISettings.diSOT2Receive > 0 AND p_tyDISettings.diSOT2Receive <= UDINT_TO_DINT(p_udiMax) THEN
					tyDInput.bSOT2Receive	:= a_bPhysicalDI[p_tyDISettings.diSOT2Receive];
				ELSE
					tyDInput.bSOT2Receive	:= FALSE;
				END_IF

				IF p_tyDISettings.diSOT2AIVError > 0 AND p_tyDISettings.diSOT2AIVError <= UDINT_TO_DINT(p_udiMax) THEN
					tyDInput.bSOT2AIVError	:= a_bPhysicalDI[p_tyDISettings.diSOT2AIVError];
				ELSE
					tyDInput.bSOT2AIVError	:= FALSE;
				END_IF

				IF p_tyDISettings.diSOT2AIVSizeLarge > 0 AND p_tyDISettings.diSOT2AIVSizeLarge <= UDINT_TO_DINT(p_udiMax) THEN
					tyDInput.bSOT2AIVSizeLarge	:= a_bPhysicalDI[p_tyDISettings.diSOT2AIVSizeLarge];
				ELSE
					tyDInput.bSOT2AIVSizeLarge	:= FALSE;
				END_IF

				IF p_tyDISettings.diSOT2AIVReady > 0 AND p_tyDISettings.diSOT2AIVReady <= UDINT_TO_DINT(p_udiMax) THEN
					tyDInput.bSOT2AIVReady	:= a_bPhysicalDI[p_tyDISettings.diSOT2AIVReady];
				ELSE
					tyDInput.bSOT2AIVReady	:= FALSE;
				END_IF

				IF p_tyDISettings.diSOT2AIVAvailable > 0 AND p_tyDISettings.diSOT2AIVAvailable <= UDINT_TO_DINT(p_udiMax) THEN
					tyDInput.bSOT2AIVAvailable	:= a_bPhysicalDI[p_tyDISettings.diSOT2AIVAvailable];
				ELSE
					tyDInput.bSOT2AIVAvailable	:= FALSE;
				END_IF

				IF p_tyDISettings.diSOT3Receive > 0 AND p_tyDISettings.diSOT3Receive <= UDINT_TO_DINT(p_udiMax) THEN
					tyDInput.bSOT3Receive	:= a_bPhysicalDI[p_tyDISettings.diSOT3Receive];
				ELSE
					tyDInput.bSOT3Receive	:= FALSE;
				END_IF

				IF p_tyDISettings.diSOT3AIVError > 0 AND p_tyDISettings.diSOT3AIVError <= UDINT_TO_DINT(p_udiMax) THEN
					tyDInput.bSOT3AIVError	:= a_bPhysicalDI[p_tyDISettings.diSOT3AIVError];
				ELSE
					tyDInput.bSOT3AIVError	:= FALSE;
				END_IF

				IF p_tyDISettings.diSOT3AIVSizeLarge > 0 AND p_tyDISettings.diSOT3AIVSizeLarge <= UDINT_TO_DINT(p_udiMax) THEN
					tyDInput.bSOT3AIVSizeLarge	:= a_bPhysicalDI[p_tyDISettings.diSOT3AIVSizeLarge];
				ELSE
					tyDInput.bSOT3AIVSizeLarge	:= FALSE;
				END_IF

				IF p_tyDISettings.diSOT3AIVReady > 0 AND p_tyDISettings.diSOT3AIVReady <= UDINT_TO_DINT(p_udiMax) THEN
					tyDInput.bSOT3AIVReady	:= a_bPhysicalDI[p_tyDISettings.diSOT3AIVReady];
				ELSE
					tyDInput.bSOT3AIVReady	:= FALSE;
				END_IF

				IF p_tyDISettings.diSOT3AIVAvailable > 0 AND p_tyDISettings.diSOT3AIVAvailable <= UDINT_TO_DINT(p_udiMax) THEN
					tyDInput.bSOT3AIVAvailable	:= a_bPhysicalDI[p_tyDISettings.diSOT3AIVAvailable];
				ELSE
					tyDInput.bSOT3AIVAvailable	:= FALSE;
				END_IF

				IF p_tyDISettings.diSOT4Receive > 0 AND p_tyDISettings.diSOT4Receive <= UDINT_TO_DINT(p_udiMax) THEN
					tyDInput.bSOT4Receive	:= a_bPhysicalDI[p_tyDISettings.diSOT4Receive];
				ELSE
					tyDInput.bSOT4Receive	:= FALSE;
				END_IF

				IF p_tyDISettings.diSOT4AIVError > 0 AND p_tyDISettings.diSOT4AIVError <= UDINT_TO_DINT(p_udiMax) THEN
					tyDInput.bSOT4AIVError	:= a_bPhysicalDI[p_tyDISettings.diSOT4AIVError];
				ELSE
					tyDInput.bSOT4AIVError	:= FALSE;
				END_IF

				IF p_tyDISettings.diSOT4AIVSizeLarge > 0 AND p_tyDISettings.diSOT4AIVSizeLarge <= UDINT_TO_DINT(p_udiMax) THEN
					tyDInput.bSOT4AIVSizeLarge	:= a_bPhysicalDI[p_tyDISettings.diSOT4AIVSizeLarge];
				ELSE
					tyDInput.bSOT4AIVSizeLarge	:= FALSE;
				END_IF

				IF p_tyDISettings.diSOT4AIVReady > 0 AND p_tyDISettings.diSOT4AIVReady <= UDINT_TO_DINT(p_udiMax) THEN
					tyDInput.bSOT4AIVReady	:= a_bPhysicalDI[p_tyDISettings.diSOT4AIVReady];
				ELSE
					tyDInput.bSOT4AIVReady	:= FALSE;
				END_IF

				IF p_tyDISettings.diSOT4AIVAvailable > 0 AND p_tyDISettings.diSOT4AIVAvailable <= UDINT_TO_DINT(p_udiMax) THEN
					tyDInput.bSOT4AIVAvailable	:= a_bPhysicalDI[p_tyDISettings.diSOT4AIVAvailable];
				ELSE
					tyDInput.bSOT4AIVAvailable	:= FALSE;
				END_IF
			ELSE
				tyDInput.bSOT1Receive	:= p_tySOTSimulate1.tyBtnInPos;
				tyDInput.bSOT1AIVError	:= p_tySOTSimulate1.tyBtnError;
				tyDInput.bSOT1AIVReady		:= p_tySOTSimulate1.tyBtnRdy;
				tyDInput.bSOT1AIVAvailable	:= p_tySOTSimulate1.tyBtnAvail;

				tyDInput.bSOT2Receive	:= p_tySOTSimulate2.tyBtnInPos;
				tyDInput.bSOT2AIVError	:= p_tySOTSimulate2.tyBtnError;
				tyDInput.bSOT2AIVReady		:= p_tySOTSimulate2.tyBtnRdy;
				tyDInput.bSOT2AIVAvailable	:= p_tySOTSimulate2.tyBtnAvail;

				tyDInput.bSOT3Receive	:= p_tySOTSimulate3.tyBtnInPos;
				tyDInput.bSOT3AIVError	:= p_tySOTSimulate3.tyBtnError;
				tyDInput.bSOT3AIVReady		:= p_tySOTSimulate3.tyBtnRdy;
				tyDInput.bSOT3AIVAvailable	:= p_tySOTSimulate3.tyBtnAvail;

				tyDInput.bSOT4Receive	:= p_tySOTSimulate4.tyBtnInPos;
				tyDInput.bSOT4AIVError	:= p_tySOTSimulate4.tyBtnError;
				tyDInput.bSOT4AIVReady		:= p_tySOTSimulate4.tyBtnRdy;
				tyDInput.bSOT4AIVAvailable	:= p_tySOTSimulate4.tyBtnAvail;
			END_IF

	ELSIF p_bLinkNtParamProjSOTSenPrep = FALSE THEN

		CASE p_eLinkAGVComProtocol OF
			McSetAGVCommOPCUA:
				IF p_bUIAGVSimulationOn = FALSE THEN
					tyDInput.bFleetManagerReady	:= p_tyTagFromMes.bActive;

					tyDInput.bSOT1Receive := TRUE;
					tyDInput.bSOT1AIVError := p_tyTagFromMes.tyTagStatOfPlatforms[1].bError;
					tyDInput.bSOT1AIVSizeLarge := p_tyTagFromMes.tyTagStatOfPlatforms[1].bSizeLarge;
					tyDInput.bSOT1AIVReady := p_tyTagFromMes.tyTagStatOfPlatforms[1].bReady;
					tyDInput.bSOT1AIVAvailable := p_tyTagFromMes.tyTagStatOfPlatforms[1].bAvailable;

					tyDInput.bSOT2Receive := TRUE;
					tyDInput.bSOT2AIVError := p_tyTagFromMes.tyTagStatOfPlatforms[2].bError;
					tyDInput.bSOT2AIVSizeLarge := p_tyTagFromMes.tyTagStatOfPlatforms[2].bSizeLarge;
					tyDInput.bSOT2AIVReady := p_tyTagFromMes.tyTagStatOfPlatforms[2].bReady;
					tyDInput.bSOT2AIVAvailable := p_tyTagFromMes.tyTagStatOfPlatforms[2].bAvailable;

					tyDInput.bSOT3Receive := TRUE;
					tyDInput.bSOT3AIVError := p_tyTagFromMes.tyTagStatOfPlatforms[3].bError;
					tyDInput.bSOT3AIVSizeLarge := p_tyTagFromMes.tyTagStatOfPlatforms[3].bSizeLarge;
					tyDInput.bSOT3AIVReady := p_tyTagFromMes.tyTagStatOfPlatforms[3].bReady;
					tyDInput.bSOT3AIVAvailable := p_tyTagFromMes.tyTagStatOfPlatforms[3].bAvailable;

					tyDInput.bSOT4Receive := TRUE;
					tyDInput.bSOT4AIVError := p_tyTagFromMes.tyTagStatOfPlatforms[4].bError;
					tyDInput.bSOT4AIVSizeLarge := p_tyTagFromMes.tyTagStatOfPlatforms[4].bSizeLarge;
					tyDInput.bSOT4AIVReady := p_tyTagFromMes.tyTagStatOfPlatforms[4].bReady;
					tyDInput.bSOT4AIVAvailable := p_tyTagFromMes.tyTagStatOfPlatforms[4].bAvailable;

				ELSE
					tyDInput.bSOT1Receive	:= p_tySOTSimulate1.tyBtnInPos;
					tyDInput.bSOT1AIVError	:= p_tySOTSimulate1.tyBtnError;
					tyDInput.bSOT1AIVReady		:= p_tySOTSimulate1.tyBtnRdy;
					tyDInput.bSOT1AIVAvailable	:= p_tySOTSimulate1.tyBtnAvail;

					tyDInput.bSOT2Receive	:= p_tySOTSimulate2.tyBtnInPos;
					tyDInput.bSOT2AIVError	:= p_tySOTSimulate2.tyBtnError;
					tyDInput.bSOT2AIVReady		:= p_tySOTSimulate2.tyBtnRdy;
					tyDInput.bSOT2AIVAvailable	:= p_tySOTSimulate2.tyBtnAvail;

					tyDInput.bSOT3Receive	:= p_tySOTSimulate3.tyBtnInPos;
					tyDInput.bSOT3AIVError	:= p_tySOTSimulate3.tyBtnError;
					tyDInput.bSOT3AIVReady		:= p_tySOTSimulate3.tyBtnRdy;
					tyDInput.bSOT3AIVAvailable	:= p_tySOTSimulate3.tyBtnAvail;

					tyDInput.bSOT4Receive	:= p_tySOTSimulate4.tyBtnInPos;
					tyDInput.bSOT4AIVError	:= p_tySOTSimulate4.tyBtnError;
					tyDInput.bSOT4AIVReady		:= p_tySOTSimulate4.tyBtnRdy;
					tyDInput.bSOT4AIVAvailable	:= p_tySOTSimulate4.tyBtnAvail;
				END_IF

			McSetAGVCommDisabled:
				tyDInput.bSOT1Receive := FALSE;
				tyDInput.bSOT1AIVError := FALSE;
				tyDInput.bSOT1AIVSizeLarge := FALSE;
				tyDInput.bSOT1AIVReady := FALSE;
				tyDInput.bSOT1AIVAvailable := FALSE;

				tyDInput.bSOT2Receive := FALSE;
				tyDInput.bSOT2AIVError := FALSE;
				tyDInput.bSOT2AIVSizeLarge := FALSE;
				tyDInput.bSOT2AIVReady := FALSE;
				tyDInput.bSOT2AIVAvailable := FALSE;

				tyDInput.bSOT3Receive := FALSE;
				tyDInput.bSOT3AIVError := FALSE;
				tyDInput.bSOT3AIVSizeLarge := FALSE;
				tyDInput.bSOT3AIVReady := FALSE;
				tyDInput.bSOT3AIVAvailable	:= FALSE;

				tyDInput.bSOT4Receive := FALSE;
				tyDInput.bSOT4AIVError := FALSE;
				tyDInput.bSOT4AIVSizeLarge := FALSE;
				tyDInput.bSOT4AIVReady := FALSE;
				tyDInput.bSOT4AIVAvailable	:= FALSE;
		END_CASE
	END_IF

	IF p_tyDISettings.diPullerExtSlwSen > 0 AND p_tyDISettings.diPullerExtSlwSen <= UDINT_TO_DINT(p_udiMax) THEN
		tyDInput.bPullerExtSlwSen	:= a_bPhysicalDI[p_tyDISettings.diPullerExtSlwSen];
	ELSE
		tyDInput.bPullerExtSlwSen	:= FALSE;
	END_IF

	IF p_tyDISettings.diPullerRetSlwSen > 0 AND p_tyDISettings.diPullerRetSlwSen <= UDINT_TO_DINT(p_udiMax) THEN
		tyDInput.bPullerRetSlwSen	:= a_bPhysicalDI[p_tyDISettings.diPullerRetSlwSen];
	ELSE
		tyDInput.bPullerRetSlwSen	:= FALSE;
	END_IF

	IF p_tyDISettings.diMtrPullerTorqueSig > 0 AND p_tyDISettings.diMtrPullerTorqueSig <= UDINT_TO_DINT(p_udiMax) THEN
		tyDInput.bMtrPullerTorqueSig	:= a_bPhysicalDI[p_tyDISettings.diMtrPullerTorqueSig];
	ELSE
		tyDInput.bMtrPullerTorqueSig	:= FALSE;
	END_IF

	IF p_tyDISettings.diMtrPullerAlmSig > 0 AND p_tyDISettings.diMtrPullerAlmSig <= UDINT_TO_DINT(p_udiMax) THEN
		tyDInput.bMtrPullerAlmSig	:= a_bPhysicalDI[p_tyDISettings.diMtrPullerAlmSig];
	ELSE
		tyDInput.bMtrPullerAlmSig	:= TRUE;
	END_IF

	IF p_tyDISettings.diPullerAntiJam > 0 AND p_tyDISettings.diPullerAntiJam <= UDINT_TO_DINT(p_udiMax) THEN
		tyDInput.bPullerAntiJam	:= a_bPhysicalDI[p_tyDISettings.diPullerAntiJam];
	ELSE
		tyDInput.bPullerAntiJam	:= TRUE;
	END_IF

	IF p_tyDISettings.diMag1SafetyBarExtRS > 0 AND p_tyDISettings.diMag1SafetyBarExtRS <= UDINT_TO_DINT(p_udiMax) THEN
		tyDInput.bMag1SafetyBarExtRS	:= a_bPhysicalDI[p_tyDISettings.diMag1SafetyBarExtRS];
	ELSE
		tyDInput.bMag1SafetyBarExtRS	:= FALSE;
	END_IF

	IF p_tyDISettings.diMag1SafetyBarRetRS > 0 AND p_tyDISettings.diMag1SafetyBarRetRS <= UDINT_TO_DINT(p_udiMax) THEN
		tyDInput.bMag1SafetyBarRetRS	:= a_bPhysicalDI[p_tyDISettings.diMag1SafetyBarRetRS];
	ELSE
		tyDInput.bMag1SafetyBarRetRS	:= FALSE;
	END_IF

	IF p_tyDISettings.diMag2SafetyBarExtRS > 0 AND p_tyDISettings.diMag2SafetyBarExtRS <= UDINT_TO_DINT(p_udiMax) THEN
		tyDInput.bMag2SafetyBarExtRS	:= a_bPhysicalDI[p_tyDISettings.diMag2SafetyBarExtRS];
	ELSE
		tyDInput.bMag2SafetyBarExtRS	:= FALSE;
	END_IF

	IF p_tyDISettings.diMag2SafetyBarRetRS > 0 AND p_tyDISettings.diMag2SafetyBarRetRS <= UDINT_TO_DINT(p_udiMax) THEN
		tyDInput.bMag2SafetyBarRetRS	:= a_bPhysicalDI[p_tyDISettings.diMag2SafetyBarRetRS];
	ELSE
		tyDInput.bMag2SafetyBarRetRS	:= FALSE;
	END_IF

	IF p_tyDISettings.diMag3SafetyBarExtRS > 0 AND p_tyDISettings.diMag3SafetyBarExtRS <= UDINT_TO_DINT(p_udiMax) THEN
		tyDInput.bMag3SafetyBarExtRS	:= a_bPhysicalDI[p_tyDISettings.diMag3SafetyBarExtRS];
	ELSE
		tyDInput.bMag3SafetyBarExtRS	:= FALSE;
	END_IF

	IF p_tyDISettings.diMag3SafetyBarRetRS > 0 AND p_tyDISettings.diMag3SafetyBarRetRS <= UDINT_TO_DINT(p_udiMax) THEN
		tyDInput.bMag3SafetyBarRetRS	:= a_bPhysicalDI[p_tyDISettings.diMag3SafetyBarRetRS];
	ELSE
		tyDInput.bMag3SafetyBarRetRS	:= FALSE;
	END_IF

	IF p_tyDISettings.diMagWidthChkSen > 0 AND p_tyDISettings.diMagWidthChkSen <= UDINT_TO_DINT(p_udiMax) THEN
		tyDInput.bMagWidthChkSen	:= a_bPhysicalDI[p_tyDISettings.diMagWidthChkSen];
	ELSE
		tyDInput.bMagWidthChkSen	:= TRUE;
	END_IF

	//curtain sensor
	IF p_tyDISettings.diCurtainSensor > 0 AND p_tyDISettings.diCurtainSensor <= UDINT_TO_DINT(p_udiMax) THEN
		tyDInput.bCurtainSensor	:= a_bPhysicalDI[p_tyDISettings.diCurtainSensor];
	ELSE
		tyDInput.bCurtainSensor	:= TRUE;
	END_IF

	IF p_tyDISettings.diBypCurtainSensorPB > 0 AND p_tyDISettings.diBypCurtainSensorPB <= UDINT_TO_DINT(p_udiMax) THEN
		tyDInput.bBypCurtainSensorPB	:= a_bPhysicalDI[p_tyDISettings.diBypCurtainSensorPB];
	ELSE
		tyDInput.bBypCurtainSensorPB	:= FALSE;
	END_IF

	IF p_tyDISettings.diCurtainSafetySig2 > 0 AND p_tyDISettings.diCurtainSafetySig2 <= UDINT_TO_DINT(p_udiMax) THEN
		tyDInput.bCurtainSafetySig2	:= a_bPhysicalDI[p_tyDISettings.diCurtainSafetySig2];
	ELSE
		tyDInput.bCurtainSafetySig2	:= FALSE;
	END_IF
	//##

	IF p_tyDISettings.diInShutterOpenRS2 > 0 AND p_tyDISettings.diInShutterOpenRS2 <= UDINT_TO_DINT(p_udiMax) THEN
		tyDInput.bInShutterOpenRS2	:= a_bPhysicalDI[p_tyDISettings.diInShutterOpenRS2];
	ELSE
		tyDInput.bInShutterOpenRS2	:= FALSE;
	END_IF

	IF p_tyDISettings.diInShutterCloseRS2 > 0 AND p_tyDISettings.diInShutterCloseRS2 <= UDINT_TO_DINT(p_udiMax) THEN
		tyDInput.bInShutterCloseRS2	:= a_bPhysicalDI[p_tyDISettings.diInShutterCloseRS2];
	ELSE
		tyDInput.bInShutterCloseRS2	:= FALSE;
	END_IF

	IF p_tyDISettings.diInShutterOpenRS3 > 0 AND p_tyDISettings.diInShutterOpenRS3 <= UDINT_TO_DINT(p_udiMax) THEN
		tyDInput.bInShutterOpenRS3	:= a_bPhysicalDI[p_tyDISettings.diInShutterOpenRS3];
	ELSE
		tyDInput.bInShutterOpenRS3	:= FALSE;
	END_IF

	IF p_tyDISettings.diInShutterCloseRS3 > 0 AND p_tyDISettings.diInShutterCloseRS3 <= UDINT_TO_DINT(p_udiMax) THEN
		tyDInput.bInShutterCloseRS3	:= a_bPhysicalDI[p_tyDISettings.diInShutterCloseRS3];
	ELSE
		tyDInput.bInShutterCloseRS3	:= FALSE;
	END_IF

	IF p_tyDISettings.diMag1FixedSideDetect > 0 AND p_tyDISettings.diMag1FixedSideDetect <= UDINT_TO_DINT(p_udiMax) THEN
		tyDInput.bMag1FixedSideDetect	:= a_bPhysicalDI[p_tyDISettings.diMag1FixedSideDetect];
	ELSE
		tyDInput.bMag1FixedSideDetect	:= FALSE;
	END_IF

	IF p_tyDISettings.diMag1RemoteSideDetect > 0 AND p_tyDISettings.diMag1RemoteSideDetect <= UDINT_TO_DINT(p_udiMax) THEN
		tyDInput.bMag1RemoteSideDetect	:= a_bPhysicalDI[p_tyDISettings.diMag1RemoteSideDetect];
	ELSE
		tyDInput.bMag1RemoteSideDetect	:= FALSE;
	END_IF

	IF p_tyDISettings.diMag2FixedSideDetect > 0 AND p_tyDISettings.diMag2FixedSideDetect <= UDINT_TO_DINT(p_udiMax) THEN
		tyDInput.bMag2FixedSideDetect	:= a_bPhysicalDI[p_tyDISettings.diMag2FixedSideDetect];
	ELSE
		tyDInput.bMag2FixedSideDetect	:= FALSE;
	END_IF

	IF p_tyDISettings.diMag2RemoteSideDetect > 0 AND p_tyDISettings.diMag2RemoteSideDetect <= UDINT_TO_DINT(p_udiMax) THEN
		tyDInput.bMag2RemoteSideDetect	:= a_bPhysicalDI[p_tyDISettings.diMag2RemoteSideDetect];
	ELSE
		tyDInput.bMag2RemoteSideDetect	:= FALSE;
	END_IF

	IF p_tyDISettings.diMag3FixedSideDetect > 0 AND p_tyDISettings.diMag3FixedSideDetect <= UDINT_TO_DINT(p_udiMax) THEN
		tyDInput.bMag3FixedSideDetect	:= a_bPhysicalDI[p_tyDISettings.diMag3FixedSideDetect];
	ELSE
		tyDInput.bMag3FixedSideDetect	:= FALSE;
	END_IF

	IF p_tyDISettings.diMag3RemoteSideDetect > 0 AND p_tyDISettings.diMag3RemoteSideDetect <= UDINT_TO_DINT(p_udiMax) THEN
		tyDInput.bMag3RemoteSideDetect	:= a_bPhysicalDI[p_tyDISettings.diMag3RemoteSideDetect];
	ELSE
		tyDInput.bMag3RemoteSideDetect	:= FALSE;
	END_IF

	//Orientation with highmagdetsen
	IF p_tyDISettings.diHighMagDetSen1 > 0 AND p_tyDISettings.diHighMagDetSen1 <= UDINT_TO_DINT(p_udiMax) THEN
		tyDInput.bHighMagDetSen1	:= a_bPhysicalDI[p_tyDISettings.diHighMagDetSen1];
	ELSE
		tyDInput.bHighMagDetSen1	:= FALSE;
	END_IF
	IF p_tyDISettings.diHighMagDetSen2 > 0 AND p_tyDISettings.diHighMagDetSen2 <= UDINT_TO_DINT(p_udiMax) THEN
		tyDInput.bHighMagDetSen2	:= a_bPhysicalDI[p_tyDISettings.diHighMagDetSen2];
	ELSE
		tyDInput.bHighMagDetSen2	:= FALSE;
	END_IF
	IF p_tyDISettings.diHighMagDetSen3 > 0 AND p_tyDISettings.diHighMagDetSen3 <= UDINT_TO_DINT(p_udiMax) THEN
		tyDInput.bHighMagDetSen3	:= a_bPhysicalDI[p_tyDISettings.diHighMagDetSen3];
	ELSE
		tyDInput.bHighMagDetSen3	:= FALSE;
	END_IF

	IF p_tyDISettings.diConvClrSen > 0 AND p_tyDISettings.diConvClrSen <= UDINT_TO_DINT(p_udiMax) THEN
		//Digital Input Filter
		fbConvClrSigFltr.tSigOnFltrTm	:= DINT_TO_TIME(p_diConvClrSenOnTm);
		fbConvClrSigFltr.tSigOffFltrTm	:= DINT_TO_TIME(p_diConvClrSenOffTm);
		fbConvClrSigFltr(bSigIn := a_bPhysicalDI[p_tyDISettings.diConvClrSen]);

		tyDInput.bConvClrSen	:= fbConvClrSigFltr.bSigOut;
	ELSE
		tyDInput.bConvClrSen	:= FALSE;
	END_IF

	//ADD
	IF p_tyDISettings.diDSSafetySig > 0 AND p_tyDISettings.diDSSafetySig <= UDINT_TO_DINT(p_udiMax) THEN
		tyDInput.bDSSafetySig	:= a_bPhysicalDI[p_tyDISettings.diDSSafetySig];;
	ELSE
		tyDInput.bDSSafetySig	:= FALSE;
	END_IF

	IF p_tyDISettings.diDSUnlockCoverSig > 0 AND p_tyDISettings.diDSUnlockCoverSig <= UDINT_TO_DINT(p_udiMax) THEN
		tyDInput.bDSUnlockCoverSig	:= a_bPhysicalDI[p_tyDISettings.diDSUnlockCoverSig];;
	ELSE
		tyDInput.bDSUnlockCoverSig	:= FALSE;
	END_IF

		//Outlet shutter2
	IF p_tyDISettings.diOutShutterOpenRS2 > 0 AND p_tyDISettings.diOutShutterOpenRS2 <= UDINT_TO_DINT(p_udiMax) THEN
		tyDInput.bOutShutterOpenRS2	:= a_bPhysicalDI[p_tyDISettings.diOutShutterOpenRS2];
	ELSE
		tyDInput.bOutShutterOpenRS2	:= FALSE;
	END_IF

	IF p_tyDISettings.diOutShutterCloseRS2 > 0 AND p_tyDISettings.diOutShutterCloseRS2 <= UDINT_TO_DINT(p_udiMax) THEN
		tyDInput.bOutShutterCloseRS2	:= a_bPhysicalDI[p_tyDISettings.diOutShutterCloseRS2];
	ELSE
		tyDInput.bOutShutterCloseRS2	:= FALSE;
	END_IF

		//Trolley
	IF p_tyDISettings.diTrolleyExtRS1 > 0 AND p_tyDISettings.diTrolleyExtRS1 <= UDINT_TO_DINT(p_udiMax) THEN
		tyDInput.bTrolleyExtRS1	:= a_bPhysicalDI[p_tyDISettings.diTrolleyExtRS1];
	ELSE
		tyDInput.bTrolleyExtRS1	:= FALSE;
	END_IF
	IF p_tyDISettings.diTrolleyExtRS2 > 0 AND p_tyDISettings.diTrolleyExtRS2 <= UDINT_TO_DINT(p_udiMax) THEN
		tyDInput.bTrolleyExtRS2	:= a_bPhysicalDI[p_tyDISettings.diTrolleyExtRS2];
	ELSE
		tyDInput.bTrolleyExtRS2	:= FALSE;
	END_IF

	IF p_tyDISettings.diTrolleyPreSen1 > 0 AND p_tyDISettings.diTrolleyPreSen1 <= UDINT_TO_DINT(p_udiMax) THEN
		//Digital Input Filter
		fbTrolley1PresentSigFltr.tSigOnFltrTm	:= DINT_TO_TIME(p_diTrolleySenOnTm); //1200ms delay (locally)
		fbTrolley1PresentSigFltr.tSigOffFltrTm	:= DINT_TO_TIME(p_diTrolleySenOffTm);
		fbTrolley1PresentSigFltr(bSigIn := a_bPhysicalDI[p_tyDISettings.diTrolleyPreSen1]);
		tyDInput.bTrolleyPreSen1	:= fbTrolley1PresentSigFltr.bSigOut;
	ELSE
		tyDInput.bTrolleyPreSen1	:= FALSE;
	END_IF
	IF p_tyDISettings.diTrolleyPreSen2 > 0 AND p_tyDISettings.diTrolleyPreSen2 <= UDINT_TO_DINT(p_udiMax) THEN
		//Digital Input Filter
		fbTrolley2PresentSigFltr.tSigOnFltrTm	:= DINT_TO_TIME(p_diTrolleySenOnTm); //1200ms delay (locally)
		fbTrolley2PresentSigFltr.tSigOffFltrTm	:= DINT_TO_TIME(p_diTrolleySenOffTm);
		fbTrolley2PresentSigFltr(bSigIn := a_bPhysicalDI[p_tyDISettings.diTrolleyPreSen2]);
		tyDInput.bTrolleyPreSen2	:= fbTrolley2PresentSigFltr.bSigOut;
	ELSE
		tyDInput.bTrolleyPreSen2	:= FALSE;
	END_IF

	IF p_tyDISettings.diSlotLckSenMag1 > 0 AND p_tyDISettings.diSlotLckSenMag1 <= UDINT_TO_DINT(p_udiMax) THEN
		tyDInput.bSlotLckSenMag1	:= a_bPhysicalDI[p_tyDISettings.diSlotLckSenMag1];
	ELSE
		tyDInput.bSlotLckSenMag1	:= FALSE;
	END_IF
	IF p_tyDISettings.diSlotLckSenMag2 > 0 AND p_tyDISettings.diSlotLckSenMag2 <= UDINT_TO_DINT(p_udiMax) THEN
		tyDInput.bSlotLckSenMag2	:= a_bPhysicalDI[p_tyDISettings.diSlotLckSenMag2];
	ELSE
		tyDInput.bSlotLckSenMag2	:= FALSE;
	END_IF

	//For Simulation Only
	IF DiagCpuIsSimulated() = TRUE THEN
		tyDInput.bSafetyRlySig			:= TRUE;
		tyDInput.bEStopSig				:= TRUE;
		tyDInput.bCoverSWSig			:= TRUE;
		tyDInput.bLifterTimingBeltSen	:= TRUE;
		tyDInput.bLifterSafetyLmtSW1	:= TRUE;
		tyDInput.bLifterSafetyLmtSW2	:= TRUE;
		tyDInput.bCurtainSafetySig2		:= TRUE;
		tyDInput.bMtrPullerAlmSig		:= TRUE;
		bSimServoEn	:= FALSE;
	END_IF

	//EStop
	IF (tyDInput.bEStopSig = FALSE) AND (eStatus1 <> Error) THEN
		eStatus1	:= Error;
		udiStatus1	:= 10000;	//Emergency SSel Button Pressed
	END_IF

	//Cover Switch
	IF (tyDInput.bCoverSWSig = FALSE) AND (eStatus2 <> Error) THEN
		eStatus2	:= Error;
		udiStatus2	:= 10001;	//Door / Conver Opened
	END_IF

	//Lifter Timing Belt
	IF (tyDInput.bLifterTimingBeltSen = FALSE) AND (eStatus3 <> Error) THEN
		eStatus3	:= Error;
		udiStatus3	:= 10002;	//Lifter Timing Belt Broken
	END_IF

	//Lifter Safety Limit Switch
	IF (tyDInput.bLifterSafetyLmtSW1 = FALSE OR tyDInput.bLifterSafetyLmtSW2 = FALSE) AND (eStatus4 <> Error) THEN
		eStatus4	:= Error;
		udiStatus4	:= 10003;	//Lifter Reached Safety Limit Switch
	END_IF

	//Safety Relay
//	fbSafetyRlyRstTm(IN := NOT(p_bRstErrSafetyRlyRst));
//	IF (tyDInput.bSafetyRlySig = FALSE) AND (eStatus5 <> Error AND eStatus1 <> Error AND eStatus2 <> Error) AND fbSafetyRlyRstTm.Q AND tyDInput.bEStopSig AND tyDInput.bCoverSWSig THEN
//		eStatus5	:= Error;
//		udiStatus5	:= 10004;	//Safety Relay Signal Off
//	END_IF

	//Curtain Sensor
//	IF tyDInput.bSafetyRlySig THEN
//		fbCurtainSafetyRstTm(IN := NOT(p_bRstCurtainSenCtrl));
//		IF (tyDInput.bCurtainSafetySig2 = FALSE) AND (eStatus6 <> Error) AND fbCurtainSafetyRstTm.Q
//			AND (p_bOpsTravLifLDBypCurtainSenCtrl <> TRUE) AND p_bRstCurtainSenCtrl =FALSE THEN	// JOHN , one pulse to reset
//			eStatus6	:= Error;
//			udiStatus6	:= 10005;	//Curtain Sensor Activated
//		END_IF
//	END_IF
	//Only For Curtain Sensor Preparation
	IF p_bCurtainSenPrep THEN
		fbCurtainSafetyRstTm(IN := NOT(p_bRstCurtainSenCtrl));
		IF (NOT tyDInput.bCurtainSafetySig2) AND (eStatus6 <> Error) AND fbCurtainSafetyRstTm.Q
			AND (p_tyDO.bBypCurtainSen = FALSE) AND p_bRstCurtainSenCtrl = FALSE THEN

			IF NOT tyDInput.bSafetyRlySig THEN
			ELSE
				eStatus6	:= Error;
				udiStatus6	:= 10005;
			END_IF
		END_IF
	END_IF

	IF p_bLinkStartupRun THEN
		fbSafetyRlyRstTm(IN := NOT(p_bRstErrSafetyRlyRst));
		IF (tyDInput.bSafetyRlySig = FALSE) AND fbSafetyRlyRstTm.Q THEN
			bSafetySigErrNoBuz	:= TRUE;
		END_IF
	ELSIF bSafetySigErrNoBuz = FALSE THEN
		fbSafetyRlyRstTm(IN := NOT(p_bRstErrSafetyRlyRst));
		IF (tyDInput.bSafetyRlySig = FALSE) AND (eStatus3 <> Error AND (eStatus2<>Error AND eStatus1<>Error)) AND fbSafetyRlyRstTm.Q AND tyDInput.bEStopSig AND tyDInput.bCoverSWSig THEN
			eStatus3	:= Error;
			udiStatus3	:= 10004; //Safety Relay Signal is Off
		END_IF
	END_IF

	//Reset Error
	IF (eStatus1 = Error) AND bRstErr THEN
		eStatus1	:= Idle;
		udiStatus1	:= 0;
	END_IF

	IF (eStatus2 = Error) AND bRstErr THEN
		eStatus2	:= Idle;
		udiStatus2	:= 0;
	END_IF

	IF (eStatus3 = Error) AND bRstErr THEN
		eStatus3	:= Idle;
		udiStatus3	:= 0;
	END_IF

	IF (eStatus4 = Error) AND bRstErr THEN
		eStatus4	:= Idle;
		udiStatus4	:= 0;
	END_IF

	IF (eStatus5 = Error) AND bRstErr THEN
		eStatus5	:= Idle;
		udiStatus5	:= 0;
	END_IF

	IF (eStatus6 = Error) AND bRstErr THEN
		eStatus6	:= Idle;
		udiStatus6	:= 0;
	END_IF
END_ACTION
```

#### Act_InitGlobal.st
```iecst
(** 2018-12-10 **)
ACTION Act_InitGlobal:

	(* Always Change If Project Change *)

	//Pass Data To Link
	p_eLinkAGVComProtocol ACCESS p_McParamAGVComProtocol;
	p_bLinkNtParamProjSOTSenPrep ACCESS p_NtParamProjSOTSenPrep;
	p_bOpsTravLifLDBypCurtainSenCtrl ACCESS p_OpsTravLifLDBypCurtainSenCtrl;
	p_bCurtainSenPrep ACCESS p_NtParamProjCurtainSenPrep;
	p_bLinkStartupRun ACCESS p_StartupRun;

	//Pass Data To Internal Use
	p_udiRstErr ACCESS p_RstErrReset;
	p_tyDISettings ACCESS p_NtParamDISettings;
	p_sProgNm ACCESS p_NtParamDIProgNm;

	p_diConvLftSenOnTm ACCESS p_McParamConvLftSenOnTm;
	p_diConvLftSenOffTm ACCESS p_McParamConvLftSenOffTm;
	p_diConvRgtSenOnTm ACCESS p_McParamConvRgtSenOnTm;
	p_diConvRgtSenOffTm ACCESS p_McParamConvRgtSenOffTm;
 	p_diMagConvEntSenOnTm ACCESS p_McParamMagConvEntrySenOnTm;
	p_diMagConvEntSenOffTm ACCESS p_McParamMagConvEntrySenOffTm;
	p_diMagConvPresentSenOnTm ACCESS p_McParamMagConvPresentSenOnTm;
	p_diMagConvPresentSenOffTm ACCESS p_McParamMagConvPresentSenOffTm;

	p_bUIAGVSimulationOn ACCESS p_UIAGVSimulationOn;
	p_tySOTSimulate1 ACCESS p_UISOTSimulationSig1;
	p_tySOTSimulate2 ACCESS p_UISOTSimulationSig2;
	p_tySOTSimulate3 ACCESS p_UISOTSimulationSig3;
	p_tySOTSimulate4 ACCESS p_UISOTSimulationSig4;

	p_tyTagFromMes ACCESS p_TagFromMes;
	p_tyDO  ACCESS p_DO;
	p_eLDMag ACCESS p_NtParamProjMag;

	p_bPullConvHvBrd ACCESS p_PullConvHvBrd;
	p_bRstErrSafetyRlyRst ACCESS p_RstErrSafetyRlyRst;
	p_bRstCurtainSenCtrl ACCESS p_UISafetyCurtainReset;
	(* Always Change If Project Change *)

END_ACTION
```

#### Act_InitLocal.st
```iecst
(** 2019-03-25 **)
ACTION Act_InitLocal:

	//Input Reference Link To Local Variable
	p_udiMax ACCESS ADR(c_udiDInputMax);
	p_udiRstErr ACCESS ADR(udiRstErr);
	p_tyDISettings ACCESS ADR(tyDISettings);
	p_sProgNm ACCESS ADR(sProgNm);

	p_diConvLftSenOnTm ACCESS ADR(diConvLftSenOnTm);
	p_diConvLftSenOffTm ACCESS ADR(diConvLftSenOffTm);
	p_diConvRgtSenOnTm ACCESS ADR(diConvRgtSenOnTm);
	p_diConvRgtSenOffTm ACCESS ADR(diConvRgtSenOffTm);
	p_diMagConvEntSenOnTm ACCESS ADR(diMagConvEntSenOnTm);
	p_diMagConvEntSenOffTm ACCESS ADR(diMagConvEntSenOffTm);
	p_diMagConvPresentSenOnTm ACCESS ADR(diMagConvPresentSenOnTm);
	p_diMagConvPresentSenOffTm ACCESS ADR(diMagConvPresentSenOffTm);
	p_diConvClrSenOnTm ACCESS ADR(diConvClrSenOnTm);
	p_diConvClrSenOffTm ACCESS ADR(diConvClrSenOffTm);
	p_diTrolleySenOnTm ACCESS ADR(diTrolleySenOnTm);
	p_diTrolleySenOffTm ACCESS ADR(diTrolleySenOffTm);

END_ACTION
```

#### Act_Link.st
```iecst
(** 2021-08-04 **)
ACTION Act_Link:

END_ACTION
```

#### Cyclic.st
```iecst
(** 2019-03-22 **)
PROGRAM _CYCLIC

	IF bInitDone = FALSE THEN
		bInitDone	:= TRUE;

		Act_InitLocal;
		Act_InitGlobal;

	ELSIF bInitialDone = FALSE THEN
		bInitialDone	:= TRUE;

		Act_Initial;

	ELSE

		Act_RstErr;
		Act_Background;
		Act_Link;
		Act_Alarm1;
		Act_Alarm2;
		Act_Alarm3;
		Act_Alarm4;
		Act_Alarm5;
		Act_Alarm6;

	END_IF

END_PROGRAM
```

#### Init.st
```iecst
(** 2019-03-22 **)
PROGRAM _INIT

	(* Always Change If Project Change *)

	//Physical Configuration
//	diMagConv1EntSenOffTm	:= 300;
//	diMagConv2EntSenOffTm	:= 300;
//	diMagConv3EntSenOffTm	:= 300;

	//Pass Address To Global Address For External Use
	//Action, State & Status

	//Alarm
	p_DIAlmData1	:= ADR(tyAlmData1);
	p_DIAlmData2	:= ADR(tyAlmData2);
	p_DIAlmData3	:= ADR(tyAlmData3);
	p_DIAlmData4	:= ADR(tyAlmData4);
	p_DIAlmData5	:= ADR(tyAlmData5);
	p_DIAlmData6	:= ADR(tyAlmData6);	//JOHN

	//Output
	p_DI					:= ADR(tyDInput);
	p_DISafetyRlySig		:= ADR(tyDInput.bSafetyRlySig);
	p_DIEStopSig			:= ADR(tyDInput.bEStopSig);
	p_DICoverSWSig			:= ADR(tyDInput.bCoverSWSig);
	p_DIDSBA				:= ADR(tyDInput.bDSBA);
	p_DIDSBB				:= ADR(tyDInput.bDSBB);
	p_DIPullerExtRS			:= ADR(tyDInput.bPullerExtRS);
	p_DIPullerRetRS			:= ADR(tyDInput.bPullerRetRS);
	p_DIPullerRotRmRS		:= ADR(tyDInput.bPullerRotRmRS);
	p_DIPullerRotHmRS		:= ADR(tyDInput.bPullerRotHmRS);
	p_DIConvLftSen			:= ADR(tyDInput.bConvLftSen);
	p_DIConvRgtSen			:= ADR(tyDInput.bConvRgtSen);
	p_DILifterTimingBeltSen	:= ADR(tyDInput.bLifterTimingBeltSen);
	p_DILifterSafetyLmtSW1	:= ADR(tyDInput.bLifterSafetyLmtSW1);
	p_DILifterSafetyLmtSW2	:= ADR(tyDInput.bLifterSafetyLmtSW2);
	p_DIMag1FixedClampRS	:= ADR(tyDInput.bMag1FixedClampRS);
	p_DIMag1FixedUnclampRS	:= ADR(tyDInput.bMag1FixedUnclampRS);
	p_DIMag1RemoteClampRS	:= ADR(tyDInput.bMag1RemoteClampRS);
	p_DIMag1RemoteUnclampRS := ADR(tyDInput.bMag1RemoteUnclampRS);
	p_DIMag2FixedClampRS	:= ADR(tyDInput.bMag2FixedClampRS);
	p_DIMag2FixedUnclampRS	:= ADR(tyDInput.bMag2FixedUnclampRS);
	p_DIMag2RemoteClampRS	:= ADR(tyDInput.bMag2RemoteClampRS);
	p_DIMag2RemoteUnclampRS	:= ADR(tyDInput.bMag2RemoteUnclampRS);
	p_DIMag3FixedClampRS	:= ADR(tyDInput.bMag3FixedClampRS);
	p_DIMag3FixedUnclampRS	:= ADR(tyDInput.bMag3FixedUnclampRS);
	p_DIMag3RemoteClampRS	:= ADR(tyDInput.bMag3RemoteClampRS);
	p_DIMag3RemoteUnclampRS	:= ADR(tyDInput.bMag3RemoteUnclampRS);
	p_DIMag4FixedClampRS	:= ADR(tyDInput.bMag4FixedClampRS);
	p_DIMag4FixedUnclampRS	:= ADR(tyDInput.bMag4FixedUnclampRS);
	p_DIMag4RemoteClampRS	:= ADR(tyDInput.bMag4RemoteClampRS);
	p_DIMag4RemoteUnclampRS	:= ADR(tyDInput.bMag4RemoteUnclampRS);
	p_DIInShutterOpenRS		:= ADR(tyDInput.bInShutterOpenRS);
	p_DIInShutterCloseRS	:= ADR(tyDInput.bInShutterCloseRS);
	p_DIOutShutterOpenRS	:= ADR(tyDInput.bOutShutterOpenRS);
	p_DIOutShutterCloseRS	:= ADR(tyDInput.bOutShutterCloseRS);
	p_DIMagPresentSen1		:= ADR(tyDInput.bMagPresentSen1);
	p_DIMagPresentSen2		:= ADR(tyDInput.bMagPresentSen2);
	p_DIMagPresentSen3		:= ADR(tyDInput.bMagPresentSen3);
	p_DIMagPresentSen4		:= ADR(tyDInput.bMagPresentSen4);
	p_DIMagConvEntSen1		:= ADR(tyDInput.bMagConvEntSen1);
	p_DIMagConvEntSen2		:= ADR(tyDInput.bMagConvEntSen2);
	p_DIMagConvEntSen3		:= ADR(tyDInput.bMagConvEntSen3);
	p_DIMagConvEntSen4		:= ADR(tyDInput.bMagConvEntSen4);
	p_DIMag1AGVInPosSen1	:= ADR(tyDInput.bMag1AGVInPosSen1);
	p_DIMag1AGVInPosSen2	:= ADR(tyDInput.bMag1AGVInPosSen2);
	p_DIMag2AGVInPosSen1	:= ADR(tyDInput.bMag2AGVInPosSen1);
	p_DIMag2AGVInPosSen2	:= ADR(tyDInput.bMag2AGVInPosSen2);
	p_DIMag3AGVInPosSen1	:= ADR(tyDInput.bMag3AGVInPosSen1);
	p_DIMag3AGVInPosSen2	:= ADR(tyDInput.bMag3AGVInPosSen2);
	p_DIMag4AGVInPosSen1	:= ADR(tyDInput.bMag4AGVInPosSen1);
	p_DIMag4AGVInPosSen2	:= ADR(tyDInput.bMag4AGVInPosSen2);
	p_DIMag1OrientChkSen1	:= ADR(tyDInput.bMag1OrientChkSen1);
	p_DIMag1OrientChkSen2	:= ADR(tyDInput.bMag1OrientChkSen2);
	p_DIMag2OrientChkSen1	:= ADR(tyDInput.bMag2OrientChkSen1);
	p_DIMag2OrientChkSen2	:= ADR(tyDInput.bMag2OrientChkSen2);
	p_DIMag3OrientChkSen1	:= ADR(tyDInput.bMag3OrientChkSen1);
	p_DIMag3OrientChkSen2	:= ADR(tyDInput.bMag3OrientChkSen2);
	p_DIMag4OrientChkSen1	:= ADR(tyDInput.bMag4OrientChkSen1);
	p_DIMag4OrientChkSen2	:= ADR(tyDInput.bMag4OrientChkSen2);
	p_DIDSWidthChkSen		:= ADR(tyDInput.bDSWidthChkSen);
	p_DIMagConvHeightSen1	:= ADR(tyDInput.bMagConvHeightSen1);
	p_DIMagConvHeightSen2	:= ADR(tyDInput.bMagConvHeightSen2);
	p_DIMagConvHeightSen3	:= ADR(tyDInput.bMagConvHeightSen3);
	p_DIMagConvHeightSen4	:= ADR(tyDInput.bMagConvHeightSen4);
	p_DIMagConvSmallMagSen1	:= ADR(tyDInput.bMagConvSmallMagSen1);
	p_DIMagConvSmallMagSen2	:= ADR(tyDInput.bMagConvSmallMagSen2);
	p_DIMagConvSmallMagSen3	:= ADR(tyDInput.bMagConvSmallMagSen3);
	p_DIMagConvSmallMagSen4	:= ADR(tyDInput.bMagConvSmallMagSen4);
	p_DIMagConvLargeMagSen1	:= ADR(tyDInput.bMagConvLargeMagSen1);
	p_DIMagConvLargeMagSen2	:= ADR(tyDInput.bMagConvLargeMagSen2);
	p_DIMagConvLargeMagSen3	:= ADR(tyDInput.bMagConvLargeMagSen3);
	p_DIMagConvLargeMagSen4	:= ADR(tyDInput.bMagConvLargeMagSen4);
	p_DIMagConvCAB717MagSen1:= ADR(tyDInput.bMagConvCAB717MagSen1);
	p_DIMagConvCAB717MagSen2:= ADR(tyDInput.bMagConvCAB717MagSen2);
	p_DIMagConvCAB717MagSen3:= ADR(tyDInput.bMagConvCAB717MagSen3);
	p_DIMagConvCAB717MagSen4:= ADR(tyDInput.bMagConvCAB717MagSen4);
	p_DIMag1SelUnclampRS	:= ADR(tyDInput.bMag1SelUnClampRS);
	p_DIMag2SelUnclampRS	:= ADR(tyDInput.bMag2SelUnClampRS);
	p_DIMag3SelUnclampRS	:= ADR(tyDInput.bMag3SelUnClampRS);
	p_DIMag4SelUnclampRS	:= ADR(tyDInput.bMag4SelUnClampRS);
	p_DISOT1Receive 		:= ADR(tyDInput.bSOT1Receive);
	p_DISOT1Error 			:= ADR(tyDInput.bSOT1AIVError);
	p_DISOT1SizeLarge		:= ADR(tyDInput.bSOT1AIVSizeLarge);
	p_DISOT1Ready			:= ADR(tyDInput.bSOT1AIVReady);
	p_DISOT1Available		:= ADR(tyDInput.bSOT1AIVAvailable);
	p_DISOT2Receive 		:= ADR(tyDInput.bSOT2Receive);
	p_DISOT2Error 			:= ADR(tyDInput.bSOT2AIVError);
	p_DISOT2SizeLarge		:= ADR(tyDInput.bSOT2AIVSizeLarge);
	p_DISOT2Ready			:= ADR(tyDInput.bSOT2AIVReady);
	p_DISOT2Available		:= ADR(tyDInput.bSOT2AIVAvailable);
	p_DISOT3Receive 		:= ADR(tyDInput.bSOT3Receive);
	p_DISOT3Error 			:= ADR(tyDInput.bSOT3AIVError);
	p_DISOT3SizeLarge		:= ADR(tyDInput.bSOT3AIVSizeLarge);
	p_DISOT3Ready			:= ADR(tyDInput.bSOT3AIVReady);
	p_DISOT3Available		:= ADR(tyDInput.bSOT3AIVAvailable);
	p_DISOT4Receive 		:= ADR(tyDInput.bSOT4Receive);
	p_DISOT4Error 			:= ADR(tyDInput.bSOT4AIVError);
	p_DISOT4SizeLarge		:= ADR(tyDInput.bSOT4AIVSizeLarge);
	p_DISOT4Ready			:= ADR(tyDInput.bSOT4AIVReady);
	p_DISOT4Available		:= ADR(tyDInput.bSOT4AIVAvailable);
	p_DIFleetManagerActive	:= ADR(tyDInput.bFleetManagerReady);
	p_DIPullerExtSlwSen		:= ADR(tyDInput.bPullerExtSlwSen);
	p_DIPullerRetSlwSen		:= ADR(tyDInput.bPullerRetSlwSen);
	p_DIMtrPullerTorqueSig	:= ADR(tyDInput.bMtrPullerTorqueSig);
	p_DIMtrPullerAlmSig		:= ADR(tyDInput.bMtrPullerAlmSig);
	p_DIMag1SafetyBarExtRS	:= ADR(tyDInput.bMag1SafetyBarExtRS);
	p_DIMag1SafetyBarRetRS	:= ADR(tyDInput.bMag1SafetyBarRetRS);
	p_DIMag2SafetyBarExtRS	:= ADR(tyDInput.bMag2SafetyBarExtRS);
	p_DIMag2SafetyBarRetRS	:= ADR(tyDInput.bMag2SafetyBarRetRS);
	p_DIMag3SafetyBarExtRS	:= ADR(tyDInput.bMag3SafetyBarExtRS);
	p_DIMag3SafetyBarRetRS	:= ADR(tyDInput.bMag3SafetyBarRetRS);
	p_DIMagWidthChkSen		:= ADR(tyDInput.bMagWidthChkSen);
	p_DIPullerAntiJamSen	:= ADR(tyDInput.bPullerAntiJam);

	p_DIInShutterOpenRS2	:= ADR(tyDInput.bInShutterOpenRS2);
	p_DIInShutterCloseRS2	:= ADR(tyDInput.bInShutterCloseRS2);
	p_DIInShutterOpenRS3	:= ADR(tyDInput.bInShutterOpenRS3);
	p_DIInShutterCloseRS3	:= ADR(tyDInput.bInShutterCloseRS3);
	p_DIMag1FixedSideDetect	:= ADR(tyDInput.bMag1FixedSideDetect);
	p_DIMag1RemoteSideDetect	:= ADR(tyDInput.bMag1RemoteSideDetect);
	p_DIMag2FixedSideDetect		:= ADR(tyDInput.bMag2FixedSideDetect);
	p_DIMag2RemoteSideDetect	:= ADR(tyDInput.bMag2RemoteSideDetect);
	p_DIMag3FixedSideDetect		:= ADR(tyDInput.bMag3FixedSideDetect);
	p_DIMag3RemoteSideDetect	:= ADR(tyDInput.bMag3RemoteSideDetect);

	p_DICurtainSen			:= ADR(tyDInput.bCurtainSensor);
	p_DIBypCurtainSensorPB	:= ADR(tyDInput.bBypCurtainSensorPB);
	p_DICurtainSafetySig2	:= ADR(tyDInput.bCurtainSafetySig2); 		// JOHN
	p_DIHighMagDetSen1		:= ADR(tyDInput.bHighMagDetSen1); 	// Detect the Magazine Height together with magazine orientation
	p_DIHighMagDetSen2		:= ADR(tyDInput.bHighMagDetSen2);	//as mag orientation sen is always detecting magazine at any orientation
	p_DIHighMagDetSen3		:= ADR(tyDInput.bHighMagDetSen3);	//For magazine without metal plate detecting
	p_DIConvClrSen			:= ADR(tyDInput.bConvClrSen); 	   //conveyor clear sensor

	p_DIDSSafetySig			:= ADR(tyDInput.bDSSafetySig);	//ADD
	p_DIDSUnlockSafetySig	:= ADR(tyDInput.bDSUnlockCoverSig); //ADD

	p_DIMcSelfTest	:= ADR(bSelfTest);
	p_DISimServoEn	:= ADR(bSimServoEn);

	p_DIOutShutterOpenRS2	:= ADR(tyDInput.bOutShutterOpenRS2);
	p_DIOutShutterCloseRS2	:= ADR(tyDInput.bOutShutterCloseRS2);

	p_DITrolleyExtRS1	:= ADR(tyDInput.bTrolleyExtRS1);
	p_DITrolleyExtRS2	:= ADR(tyDInput.bTrolleyExtRS2);
	p_DITrolleyPreSen1	:= ADR(tyDInput.bTrolleyPreSen1);
	p_DITrolleyPreSen2	:= ADR(tyDInput.bTrolleyPreSen2);
	p_DISlotLckSenMag1	:= ADR(tyDInput.bSlotLckSenMag1);
	p_DISlotLckSenMag2	:= ADR(tyDInput.bSlotLckSenMag2);

	(* Always Change If Project Change *)

END_PROGRAM
```

### DOutput.typ
```iecst
(*2018-12-13*)
(**)
(*Action*)

TYPE
	eDOAction :
		(
		DOActIdle,
		DOActRstAll,
		DOActSetBypassCoverSwitch,
		DOActRstBypassCoverSwitch
		);
END_TYPE

(**)
(*Data*)

TYPE
	tyDigitalOutput : 	STRUCT
		bSafetyRlyRst : BOOL;
		bTLRed : BOOL;
		bTLAmber : BOOL;
		bTLGreen : BOOL;
		bBuzzer : BOOL;
		bDBAA : BOOL;
		bDBAB : BOOL;
		bPullerExtCtrl : BOOL;
		bPullerRetCtrl : BOOL;
		bRotPullerCtrl : BOOL;
		bMag1FixedClampCtrl : BOOL;
		bMag1RemoteClampCtrl : BOOL;
		bMag2FixedClampCtrl : BOOL;
		bMag2RemoteClampCtrl : BOOL;
		bMag3FixedClampCtrl : BOOL;
		bMag3RemoteClampCtrl : BOOL;
		bMag4FixedClampCtrl : BOOL;
		bMag4RemoteClampCtrl : BOOL;
		bInShutterOpenCtrl : BOOL;
		bInShutterCloseCtrl : BOOL;
		bOutShutterOpenCtrl : BOOL;
		bOutShutterCloseCtrl : BOOL;
		bMag1ConvMtrIn : BOOL;
		bMag1ConvMtrOut : BOOL;
		bMag2ConvMtrIn : BOOL;
		bMag2ConvMtrOut : BOOL;
		bMag3ConvMtrIn : BOOL;
		bMag3ConvMtrOut : BOOL;
		bMag4ConvMtrIn : BOOL;
		bMag4ConvMtrOut : BOOL;
		bPullConvMtrOn : BOOL;
		bMag1SelClampCtrl : BOOL;
		bMag2SelClampCtrl : BOOL;
		bMag3SelClampCtrl : BOOL;
		bMag4SelClampCtrl : BOOL;
		bSOT1MagError : BOOL;
		bSOT1MagSizeLarge : BOOL;
		bSOT1MagReady : BOOL;
		bSOT1MagAvailable : BOOL;
		bSOT2MagError : BOOL;
		bSOT2MagSizeLarge : BOOL;
		bSOT2MagReady : BOOL;
		bSOT2MagAvailable : BOOL;
		bSOT3MagError : BOOL;
		bSOT3MagSizeLarge : BOOL;
		bSOT3MagReady : BOOL;
		bSOT3MagAvailable : BOOL;
		bSOT4MagError : BOOL;
		bSOT4MagSizeLarge : BOOL;
		bSOT4MagReady : BOOL;
		bSOT4MagAvailable : BOOL;
		bMag1ReqToBring : BOOL;
		bMag1ReqToGet : BOOL;
		bMag2ReqToBring : BOOL;
		bMag2ReqToGet : BOOL;
		bMag3ReqToBring : BOOL;
		bMag3ReqToGet : BOOL;
		bMag4ReqToBring : BOOL;
		bMag4ReqToGet : BOOL;
		bUSBRun : BOOL;
		bMtrPshrExt : BOOL;
		bMtrPshrRet : BOOL;
		bMtrPshrOn : BOOL;
		bMtrPshrBrakeRls : BOOL;
		bMtrPshrSpdBinBit0 : BOOL;
		bMtrPshrSpdBinBit1 : BOOL;
		bMtrPshrSpdBinBit2 : BOOL;
		bMtrPshrAlmRst : BOOL;
		bMag1SafetyBarRetCtrl : BOOL;
		bMag2SafetyBarRetCtrl : BOOL;
		bMag3SafetyBarRetCtrl : BOOL;
		bBypCurtainSen : BOOL;
		bRstCurtainSen : BOOL;
		bInShutterOpenCtrl2 : BOOL;
		bInShutterCloseCtrl2 : BOOL;
		bInShutterOpenCtrl3 : BOOL;
		bInShutterCloseCtrl3 : BOOL;
		bMag1FixedClampOpenCtrl : BOOL;
		bMag1RemoteClampOpenCtrl : BOOL;
		bMag2FixedClampOpenCtrl : BOOL;
		bMag2RemoteClampOpenCtrl : BOOL;
		bMag3FixedClampOpenCtrl : BOOL;
		bMag3RemoteClampOpenCtrl : BOOL;
		bMcSafetySigToDS : BOOL;
		bOutShutterOpenCtrl2 : BOOL;
		bOutShutterCloseCtrl2 : BOOL;
		bTrolleyLckCtrl1 : BOOL;
		bTrolleyLckCtrl2 : BOOL;
		bSPARE15 : BOOL;
		bSPARE16 : BOOL;
		bSPARE17 : BOOL;
		bSPARE18 : BOOL;
		bSPARE19 : BOOL;
		bSPARE20 : BOOL;
	END_STRUCT;
	tyDigitalOutputSettings : 	STRUCT
		diSafetyRlyRst : DINT;
		diTLRed : DINT;
		diTLAmber : DINT;
		diTLGreen : DINT;
		diBuzzer : DINT;
		diDBAA : DINT;
		diDBAB : DINT;
		diPullerExtCtrl : DINT;
		diPullerRetCtrl : DINT;
		diRotPullerCtrl : DINT;
		diMag1FixedClampCtrl : DINT;
		diMag1RemoteClampCtrl : DINT;
		diMag2FixedClampCtrl : DINT;
		diMag2RemoteClampCtrl : DINT;
		diMag3FixedClampCtrl : DINT;
		diMag3RemoteClampCtrl : DINT;
		diMag4FixedClampCtrl : DINT;
		diMag4RemoteClampCtrl : DINT;
		diInShutterOpenCtrl : DINT;
		diInShutterCloseCtrl : DINT;
		diOutShutterOpenCtrl : DINT;
		diOutShutterCloseCtrl : DINT;
		diMag1ConvMtrIn : DINT;
		diMag1ConvMtrOut : DINT;
		diMag2ConvMtrIn : DINT;
		diMag2ConvMtrOut : DINT;
		diMag3ConvMtrIn : DINT;
		diMag3ConvMtrOut : DINT;
		diMag4ConvMtrIn : DINT;
		diMag4ConvMtrOut : DINT;
		diPullConvMtrOn : DINT;
		diMag1SelClampCtrl : DINT;
		diMag2SelClampCtrl : DINT;
		diMag3SelClampCtrl : DINT;
		diMag4SelClampCtrl : DINT;
		diSOT1MagError : DINT;
		diSOT1MagSizeLarge : DINT;
		diSOT1MagReady : DINT;
		diSOT1MagAvailable : DINT;
		diSOT2MagError : DINT;
		diSOT2MagSizeLarge : DINT;
		diSOT2MagReady : DINT;
		diSOT2MagAvailable : DINT;
		diSOT3MagError : DINT;
		diSOT3MagSizeLarge : DINT;
		diSOT3MagReady : DINT;
		diSOT3MagAvailable : DINT;
		diSOT4MagError : DINT;
		diSOT4MagSizeLarge : DINT;
		diSOT4MagReady : DINT;
		diSOT4MagAvailable : DINT;
		diMag1ReqToBring : DINT;
		diMag1ReqToGet : DINT;
		diMag2ReqToBring : DINT;
		diMag2ReqToGet : DINT;
		diMag3ReqToBring : DINT;
		diMag3ReqToGet : DINT;
		diMag4ReqToBring : DINT;
		diMag4ReqToGet : DINT;
		diUSBRun : DINT;
		diMtrPshrExt : DINT;
		diMtrPshrRet : DINT;
		diMtrPshrOn : DINT;
		diMtrPshrBrakeRls : DINT;
		diMtrPshrSpdBinBit0 : DINT;
		diMtrPshrSpdBinBit1 : DINT;
		diMtrPshrSpdBinBit2 : DINT;
		diMtrPshrAlmRst : DINT;
		diMag1SafetyBarRetCtrl : DINT;
		diMag2SafetyBarRetCtrl : DINT;
		diMag3SafetyBarRetCtrl : DINT;
		diBypCurtainSen : DINT;
		diBypCurtainSensorPBLED : DINT;
		diRstCurtainSen : DINT;
		diInShutterOpenCtrl2 : DINT;
		diInShutterCloseCtrl2 : DINT;
		diInShutterOpenCtrl3 : DINT;
		diInShutterCloseCtrl3 : DINT;
		diMag1FixedClampOpenCtrl : DINT;
		diMag1RemoteClampOpenCtrl : DINT;
		diMag2FixedClampOpenCtrl : DINT;
		diMag2RemoteClampOpenCtrl : DINT;
		diMag3FixedClampOpenCtrl : DINT;
		diMag3RemoteClampOpenCtrl : DINT;
		diMag4FixedClampOpenCtrl : DINT;
		diMag4RemoteClampOpenCtrl : DINT;
		diMcSafetySigToDS : DINT;
		diOutShutterOpenCtrl2 : DINT;
		diOutShutterCloseCtrl2 : DINT;
		diTrolleyLckCtrl1 : DINT;
		diTrolleyLckCtrl2 : DINT;
		diSPARE15 : DINT;
		diSPARE16 : DINT;
		diSPARE17 : DINT;
		diSPARE18 : DINT;
		diSPARE19 : DINT;
		diSPARE20 : DINT;
	END_STRUCT;
END_TYPE
```

### DOutput.var
```iecst
(*2019-01-08*)
(**)
(*Constant*)
VAR CONSTANT
	c_udiDOutputMax : UDINT := 300; (*Constant Digital Output Quantity (+1 For Damaged)(+1 For Spare)*)
END_VAR
(**)
(*Action & State & Status*)
VAR
	p_DOStat : UDINT;
	p_DOStatus : UDINT;
	p_DOStatTxt : UDINT;
END_VAR
(**)
(*Alarm*)
(**)
(*Output*)
VAR
	p_DO : UDINT;
END_VAR
```

### Program Logical/DOutput/DOutput (IEC, version 1.00.0)

#### Act_InitGlobal.st - Change By Project
```iecst
(** 2019-05-20 **)
ACTION Act_InitGlobal:

	(* Always Change If Project Change *)

	//Pass Data To Link
	p_bLinkOpsRun ACCESS p_OpsRun;
	p_bLinkPullerExtCtrl ACCESS p_Pneu2SenPullerExtCtrl;
	p_bLinkPullerRetCtrl ACCESS p_Pneu2SenPullerRetCtrl;
	p_bLinkPullConvExtCtrl ACCESS p_PullConvPullerExtCtrl;
	p_bLinkPullConvRetCtrl ACCESS p_PullConvPullerRetCtrl;
	p_eLinkAGVComProtocol ACCESS p_McParamAGVComProtocol;
	p_bLinkNtParamProjSOTSenPrep ACCESS p_NtParamProjSOTSenPrep;

	p_bLinkAGVCommRdy1 ACCESS p_OpsMagConvLD1AGVCommRdy;
	p_bLinkAGVCommRdy2 ACCESS p_OpsMagConvLD2AGVCommRdy;
	p_bLinkAGVCommRdy3 ACCESS p_OpsMagConvLD3AGVCommRdy;
	p_bLinkOpsBypCurtainLED ACCESS p_OpsTravLifLDBypCurtainLED;	//Bypass Curtain Push Button LED
	p_bLinkOpsBypCurtainSen ACCESS p_OpsTravLifLDBypCurtainSenCtrl; //Bypass the Curtain Sensor
	p_eNtParamCustomerReq ACCESS p_NtParamCustomerReq;

	//Pass Data To Internal Use
	p_eAct ACCESS p_UIDOAct;
	p_tyDOSettings ACCESS p_NtParamDOSettings;
	p_bManual ACCESS p_UIUIMnlMod;
	p_bSafetyRlyRst ACCESS p_RstErrSafetyRlyRst;

	p_bTLRed ACCESS p_TLBuzRed;
//	p_bTLAmber ACCESS p_TLBuzAmber; //For Job 2023-0061
//	p_bTLAmber ACCESS p_TLBuzWhite;
	p_bTLGreen ACCESS p_TLBuzGreen;
	p_bBuzzer ACCESS p_TLBuzBeep;
	p_bDBAA ACCESS p_DSSMEMAADBA;
	p_bDBAB ACCESS p_DSSMEMABDBA;
	p_bRotPullerCtrl ACCESS p_PullConvRotRemoteCtrl;
	p_bMag1FixedClampCtrl ACCESS p_MagConv2Clp1FixClprClampCtrl;
	p_bMag1RemoteClampCtrl ACCESS p_MagConv2Clp1RmtClprClampCtrl;
	p_bMag2FixedClampCtrl ACCESS p_MagConv2Clp2FixClprClampCtrl;
	p_bMag2RemoteClampCtrl ACCESS p_MagConv2Clp2RmtClprClampCtrl;
	p_bMag3FixedClampCtrl ACCESS p_MagConv2Clp3FixClprClampCtrl;
	p_bMag3RemoteClampCtrl ACCESS p_MagConv2Clp3RmtClprClampCtrl;
	p_bMag4FixedClampCtrl ACCESS p_MagConv2Clp4FixClprClampCtrl;
	p_bMag4RemoteClampCtrl ACCESS p_MagConv2Clp4RmtClprClampCtrl;

	p_bMag1FixedClampOpenCtrl ACCESS p_MagConv2Clp1FixClprClampCtrl;
	p_bMag1RemoteClampOpenCtrl ACCESS p_MagConv2Clp1RmtClprClampCtrl;
	p_bMag2FixedClampOpenCtrl ACCESS p_MagConv2Clp2FixClprClampCtrl;
	p_bMag2RemoteClampOpenCtrl ACCESS p_MagConv2Clp2RmtClprClampCtrl;
	p_bMag3FixedClampOpenCtrl ACCESS p_MagConv2Clp3FixClprClampCtrl;
	p_bMag3RemoteClampOpenCtrl ACCESS p_MagConv2Clp3RmtClprClampCtrl;

	p_bInShutterOpenCtrl ACCESS p_Pneu2SenInShutterRetCtrl;
	p_bInShutterCloseCtrl ACCESS p_Pneu2SenInShutterExtCtrl;
	p_bOutShutterOpenCtrl ACCESS p_Pneu2SenOutShutterRetCtrl;
	p_bOutShutterCloseCtrl ACCESS p_Pneu2SenOutShutterExtCtrl;
	p_bMag1ConvMtrIn ACCESS p_MagConv2Clp1MtrSigOnOrLToR;
	p_bMag1ConvMtrOut ACCESS p_MagConv2Clp1MtrDirOrRToL;
	p_bMag2ConvMtrIn ACCESS p_MagConv2Clp2MtrSigOnOrLToR;
	p_bMag2ConvMtrOut ACCESS p_MagConv2Clp2MtrDirOrRToL;
	p_bMag3ConvMtrIn ACCESS p_MagConv2Clp3MtrSigOnOrLToR;
	p_bMag3ConvMtrOut ACCESS p_MagConv2Clp3MtrDirOrRToL;
	p_bMag4ConvMtrIn ACCESS p_MagConv2Clp4MtrSigOnOrLToR;
	p_bMag4ConvMtrOut ACCESS p_MagConv2Clp4MtrDirOrRToL;
	p_bPullConvMtrOn ACCESS p_PullConvMtrSigOnOrLToR;
	p_bMag1SelClampCtrl ACCESS p_PneuNoSenSelClamp1RetCtrl;
	p_bMag2SelClampCtrl ACCESS p_PneuNoSenSelClamp2RetCtrl;
	p_bMag3SelClampCtrl ACCESS p_PneuNoSenSelClamp3RetCtrl;
	p_bMag4SelClampCtrl ACCESS p_PneuNoSenSelClamp4RetCtrl;
	p_bUSBRun	ACCESS	p_UIUSBRun;

	p_bMtrPshrExt ACCESS p_MtrPshrCW;
	p_bMtrPshrRet ACCESS p_MtrPshrCCW;
	p_bMtrPshrOn ACCESS p_MtrPshrSigOn;
	p_bMtrPshrBrakeRls ACCESS p_MtrPshrBrake;
	p_bMtrPshrSpdBinBit0 ACCESS p_MtrPshrSpdBinBit0;
	p_bMtrPshrSpdBinBit1 ACCESS p_MtrPshrSpdBinBit1;
	p_bMtrPshrSpdBinBit2 ACCESS p_MtrPshrSpdBinBit2;
	p_bMtrPshrAlmRst ACCESS p_MtrPshrAlmRst;

	p_bMag1SafetyBarRetCtrl ACCESS p_Pneu2SMag1SafetyBarRetCtrl;
	p_bMag2SafetyBarRetCtrl ACCESS p_Pneu2SMag2SafetyBarRetCtrl;
	p_bMag3SafetyBarRetCtrl ACCESS p_Pneu2SMag3SafetyBarRetCtrl;

	p_bInShutterOpenCtrl2 ACCESS p_Pneu2SenInShutterRetCtrl2;
	p_bInShutterCloseCtrl2 ACCESS p_Pneu2SenInShutterExtCtrl2;
	p_bInShutterOpenCtrl3 ACCESS p_Pneu2SenInShutterRetCtrl3;
	p_bInShutterCloseCtrl3 ACCESS p_Pneu2SenInShutterExtCtrl3;

//	p_bBypCurtainSensorPBLED ACCESS p_OpsTravLifLDBypCurtainLED;	//JOHN
//	p_bBypCurtainSenCtrl ACCESS p_OpsTravLifLDBypCurtainSenCtrl; //JOHN
	p_bUIMachineSafetySigToDS ACCESS p_UIMachineSafetySigToDS; //ADD

	p_bOutShutterOpenCtrl2 ACCESS p_Pneu2SenOutShutterRetCtrl2;
	p_bOutShutterCloseCtrl2 ACCESS p_Pneu2SenOutShutterExtCtrl2;

	p_bTrolleyExtCtrl ACCESS p_PneuExtSenTrllyExtCtrl;
	p_bTrolleyExtCtrl2 ACCESS p_PneuExtSenTrlly2ExtCtrl;
	(* Always Change If Project Change *)

END_ACTION
```

#### InputRef_Link.var - Change By Project
```iecst
(*2019-04-09*)
(**)
(*External Data*)
VAR
	p_bLinkPullerExtCtrl : REFERENCE TO BOOL;
	p_bLinkPullerRetCtrl : REFERENCE TO BOOL;
	p_bLinkPullConvExtCtrl : REFERENCE TO BOOL;
	p_bLinkPullConvRetCtrl : REFERENCE TO BOOL;
	p_eLinkAGVComProtocol : REFERENCE TO eMcAGVCommProtocol;
	p_bLinkNtParamProjSOTSenPrep : REFERENCE TO BOOL;
	p_bLinkOpsRun : REFERENCE TO BOOL;
END_VAR
(*For curtain seq*)
VAR
	p_bLinkAGVCommRdy1 : REFERENCE TO BOOL;
	p_bLinkAGVCommRdy2 : REFERENCE TO BOOL;
	p_bLinkAGVCommRdy3 : REFERENCE TO BOOL;
	p_bLinkOpsBypCurtainSen : REFERENCE TO BOOL;
	p_bLinkOpsBypCurtainLED : REFERENCE TO BOOL;
	p_eNtParamCustomerReq : REFERENCE TO eCustomer;
END_VAR
```

#### Act_Link.st - Change By Project
```iecst
(** 2019-05-20 **)
ACTION Act_Link:
	IF p_eNtParamCustomerReq = Siemens THEN
		p_bTLAmber ACCESS p_TLBuzWhite;
	ELSE
		p_bTLAmber ACCESS p_TLBuzAmber;
	END_IF

	p_bPullerExtCtrl	:= p_bLinkPullerExtCtrl OR p_bLinkPullConvExtCtrl;
	p_bPullerRetCtrl	:= p_bLinkPullerRetCtrl OR p_bLinkPullConvRetCtrl;

	IF p_bManual THEN

		p_bSOTMagError1	ACCESS p_UISOTMagErr1;
		p_bSOTMagError2	ACCESS p_UISOTMagErr2;
		p_bSOTMagError3	ACCESS p_UISOTMagErr3;
		p_bSOTMagError4	ACCESS p_UISOTMagErr4;
		p_bSOTMagReady1	ACCESS p_UISOTMagRdy1;
		p_bSOTMagReady2	ACCESS p_UISOTMagRdy2;
		p_bSOTMagReady3	ACCESS p_UISOTMagRdy3;
		p_bSOTMagReady4	ACCESS p_UISOTMagRdy4;
		p_bSOTMagAvailable1	ACCESS p_UISOTMagAvail1;
		p_bSOTMagAvailable2	ACCESS p_UISOTMagAvail2;
		p_bSOTMagAvailable3	ACCESS p_UISOTMagAvail3;
		p_bSOTMagAvailable4	ACCESS p_UISOTMagAvail4;
		p_bSOTMagSizeLarge1	ACCESS p_UISOTMagSLarge1;
		p_bSOTMagSizeLarge2	ACCESS p_UISOTMagSLarge2;
		p_bSOTMagSizeLarge3 ACCESS p_UISOTMagSLarge3;
		p_bSOTMagSizeLarge4	ACCESS p_UISOTMagSLarge4;

		p_bRequestToBring1 ACCESS p_UIAIVReqBring1;
		p_bRequestToBring2 ACCESS p_UIAIVReqBring2;
		p_bRequestToBring3 ACCESS p_UIAIVReqBring3;
		p_bRequestToBring4 ACCESS p_UIAIVReqBring4;

		p_bRequestToGet1 ACCESS p_UIAIVReqGet1;
		p_bRequestToGet2 ACCESS p_UIAIVReqGet2;
		p_bRequestToGet3 ACCESS p_UIAIVReqGet3;
		p_bRequestToGet4 ACCESS p_UIAIVReqGet4;

	ELSIF p_bLinkOpsRun THEN

		p_bSOTMagReady1 ACCESS p_USSOT1USB;
		p_bSOTMagReady2 ACCESS p_USSOT2USB;
		p_bSOTMagReady3 ACCESS p_USSOT3USB;
		p_bSOTMagReady4 ACCESS p_USSOT4USB;

		p_bSOTMagError1 ACCESS p_AlarmErr;
		p_bSOTMagError2 ACCESS p_AlarmErr;
		p_bSOTMagError3 ACCESS p_AlarmErr;
		p_bSOTMagError4 ACCESS p_AlarmErr;

		p_bSOTMagAvailable1 ACCESS p_DSSOT1DBA;
		p_bSOTMagAvailable2 ACCESS p_DSSOT2DBA;
		p_bSOTMagAvailable3 ACCESS p_DSSOT3DBA;
		p_bSOTMagAvailable4 ACCESS p_DSSOT4DBA;

		p_bSOTMagSizeLarge1 ACCESS p_DSSOT1MagSizeLarge;
		p_bSOTMagSizeLarge2 ACCESS p_DSSOT2MagSizeLarge;
		p_bSOTMagSizeLarge3 ACCESS p_DSSOT3MagSizeLarge;
		p_bSOTMagSizeLarge4 ACCESS p_DSSOT4MagSizeLarge;

		p_bRequestToBring1 ACCESS p_Buffer1MagRemoved;
		p_bRequestToBring2 ACCESS p_Buffer2MagRemoved;
		p_bRequestToBring3 ACCESS p_Buffer3MagRemoved;
		p_bRequestToBring4 ACCESS p_Buffer4MagRemoved;

		p_bRequestToGet1 ACCESS p_DSSOT1DBA;
		p_bRequestToGet2 ACCESS p_DSSOT2DBA;
		p_bRequestToGet3 ACCESS p_DSSOT3DBA;
		p_bRequestToGet4 ACCESS p_DSSOT4DBA;

	ELSE
		p_bSOTMagReady1 := FALSE;
		p_bSOTMagReady2 := FALSE;
		p_bSOTMagReady3 := FALSE;
		p_bSOTMagReady4 := FALSE;

		p_bSOTMagError1 ACCESS p_AlarmErr;
		p_bSOTMagError2 ACCESS p_AlarmErr;
		p_bSOTMagError3 ACCESS p_AlarmErr;
		p_bSOTMagError4 ACCESS p_AlarmErr;

		p_bSOTMagAvailable1 := FALSE;
		p_bSOTMagAvailable2 := FALSE;
		p_bSOTMagAvailable3 := FALSE;
		p_bSOTMagAvailable4 := FALSE;

		p_bSOTMagSizeLarge1 := FALSE;
		p_bSOTMagSizeLarge2 := FALSE;
		p_bSOTMagSizeLarge3 := FALSE;
		p_bSOTMagSizeLarge4 := FALSE;

		p_bRequestToBring1 := FALSE;
		p_bRequestToBring2 := FALSE;
		p_bRequestToBring3 := FALSE;
		p_bRequestToBring4 := FALSE;

		p_bRequestToGet1 := FALSE;
		p_bRequestToGet2 := FALSE;
		p_bRequestToGet3 := FALSE;
		p_bRequestToGet4 := FALSE;
	END_IF

	CASE p_eLinkAGVComProtocol OF
		McSetAGVCommOPCUA, McSetAGVCommDisabled:
			IF p_bLinkNtParamProjSOTSenPrep THEN
				bAgvComIODisabled := FALSE;
			ELSE
				bAgvComIODisabled := TRUE;
			END_IF

		McSetAGVCommHardIO:
				bAgvComIODisabled := FALSE;

	END_CASE

	IF p_bManual THEN
		p_bBypCurtainSen ACCESS p_UIMnlBypCurtainSen;    //byp
//		p_bBypCurtainSen ACCESS p_DIBypCurtainSensorPB;
		p_bRstCurtainSen ACCESS p_UISafetyCurtainReset;  //reset rly
		p_bBypCurtainPBLED ACCESS p_UIMnlBypCurtainPBLED;	//pb led

	ELSIF p_bLinkOpsRun THEN

		IF p_bLinkOpsBypCurtainSen OR p_bLinkAGVCommRdy1 OR p_bLinkAGVCommRdy2 OR p_bLinkAGVCommRdy3 THEN
			p_bBypCurtainSen     := TRUE;
			p_bBypCurtainPBLED	 := p_bLinkOpsBypCurtainLED;
		ELSE
			p_bBypCurtainSen	 := FALSE;
			p_bBypCurtainPBLED	 := p_bLinkOpsBypCurtainLED;
		END_IF

//		p_bBypCurtainPBLED ACCESS p_OpsTravLifLDBypCurtainLED;	//JOHN
//		p_bBypCurtainSenCtrl ACCESS p_OpsTravLifLDBypCurtainSenCtrl; //JOHN

	ELSE //stop
		p_bRstCurtainSen ACCESS p_UISafetyCurtainReset;
		p_bBypCurtainSen ACCESS p_UIMnlBypCurtainSen;//ADR(bBypCurtainSen);
		p_bBypCurtainPBLED ACCESS p_UIMnlBypCurtainPBLED;//ADR(bBypCurtainPBLED);
	END_IF

END_ACTION
```

#### Act_InitLocal.st - Change By Project
```iecst
(** 2019-03-25 **)
ACTION Act_InitLocal:

	//Input Reference Link To Local Variable
	p_udiMax ACCESS ADR(c_udiDOutputMax);
	p_eAct ACCESS ADR(eAct);
	p_tyDOSettings ACCESS ADR(tyDOSettings);
	p_bManual ACCESS ADR(bManual);

	p_bSafetyRlyRst ACCESS ADR(bSafetyRlyRst);
	p_bTLRed ACCESS ADR(bTLRed);
	p_bTLAmber ACCESS ADR(bTLAmber);
	p_bTLGreen ACCESS ADR(bTLGreen);
	p_bBuzzer ACCESS ADR(bBuzzer);
	p_bDBAA ACCESS ADR(bDBAA);
	p_bDBAB ACCESS ADR(bDBAB);
	p_bPullerExtCtrl ACCESS ADR(bPullerExtCtrl);
	p_bPullerRetCtrl ACCESS ADR(bPullerRetCtrl);
	p_bRotPullerCtrl ACCESS ADR(bRotPullerCtrl);
	p_bMag1FixedClampCtrl ACCESS ADR(bMag1FixedClampCtrl);
	p_bMag1RemoteClampCtrl ACCESS ADR(bMag1RemoteClampCtrl);
	p_bMag2FixedClampCtrl ACCESS ADR(bMag2FixedClampCtrl);
	p_bMag2RemoteClampCtrl ACCESS ADR(bMag2RemoteClampCtrl);
	p_bMag3FixedClampCtrl ACCESS ADR(bMag3FixedClampCtrl);
	p_bMag3RemoteClampCtrl ACCESS ADR(bMag3RemoteClampCtrl);
	p_bMag1FixedClampOpenCtrl ACCESS ADR (bMag1FixedClampOpenCtrl);
	p_bMag1RemoteClampOpenCtrl ACCESS ADR (bMag1RemoteClampOpenCtrl);
	p_bMag2FixedClampOpenCtrl ACCESS ADR (bMag2FixedClampOpenCtrl);
	p_bMag2RemoteClampOpenCtrl ACCESS ADR (bMag2RemoteClampOpenCtrl);
	p_bMag3FixedClampOpenCtrl ACCESS ADR (bMag3FixedClampOpenCtrl);
	p_bMag3RemoteClampOpenCtrl ACCESS ADR (bMag3RemoteClampOpenCtrl);
	p_bInShutterOpenCtrl ACCESS ADR(bInShutterOpenCtrl);
	p_bInShutterCloseCtrl ACCESS ADR(bInShutterCloseCtrl);
	p_bOutShutterOpenCtrl ACCESS ADR(bOutShutterOpenCtrl);
	p_bOutShutterCloseCtrl ACCESS ADR(bOutShutterCloseCtrl);
	p_bMag1ConvMtrIn ACCESS ADR(bMag1ConvMtrIn);
	p_bMag1ConvMtrOut ACCESS ADR(bMag1ConvMtrOut);
	p_bMag2ConvMtrIn ACCESS ADR(bMag2ConvMtrIn);
	p_bMag2ConvMtrOut ACCESS ADR(bMag2ConvMtrOut);
	p_bMag3ConvMtrIn ACCESS ADR(bMag3ConvMtrIn);
	p_bMag3ConvMtrOut ACCESS ADR(bMag3ConvMtrOut);
	p_bPullConvMtrOn ACCESS ADR(bPullConvMtrOn);
	p_bMag1SelClampCtrl ACCESS ADR(bMag1SelClampCtrl);
	p_bMag2SelClampCtrl ACCESS ADR(bMag2SelClampCtrl);
	p_bMag3SelClampCtrl ACCESS ADR(bMag3SelClampCtrl);
	p_bSOTMagError1 ACCESS ADR(bSOTMagError1);
	p_bSOTMagError2 ACCESS ADR(bSOTMagError2);
	p_bSOTMagError3 ACCESS ADR(bSOTMagError3);
	p_bSOTMagError4 ACCESS ADR(bSOTMagError4);
	p_bSOTMagReady1 ACCESS ADR(bSOTMagReady1);
	p_bSOTMagReady2 ACCESS ADR(bSOTMagReady2);
	p_bSOTMagReady3 ACCESS ADR(bSOTMagReady3);
	p_bSOTMagReady4 ACCESS ADR(bSOTMagReady4);
	p_bSOTMagAvailable1 ACCESS ADR(bSOTMagAvailable1);
	p_bSOTMagAvailable2 ACCESS ADR(bSOTMagAvailable2);
	p_bSOTMagAvailable3 ACCESS ADR(bSOTMagAvailable3);
	p_bSOTMagAvailable4 ACCESS ADR(bSOTMagAvailable4);
	p_bSOTMagSizeLarge1 ACCESS ADR(bSOTMagSLarge1);
	p_bSOTMagSizeLarge2 ACCESS ADR(bSOTMagSLarge2);
	p_bSOTMagSizeLarge3 ACCESS ADR(bSOTMagSLarge3);
	p_bSOTMagSizeLarge4 ACCESS ADR(bSOTMagSLarge4);
	p_bRequestToBring1 ACCESS ADR(bRequestToBring1);
	p_bRequestToGet1 ACCESS ADR(bRequestToGet1);
	p_bRequestToBring2 ACCESS ADR(bRequestToBring2);
	p_bRequestToGet2 ACCESS ADR(bRequestToGet2);
	p_bRequestToBring3 ACCESS ADR(bRequestToBring3);
	p_bRequestToGet3 ACCESS ADR(bRequestToGet3);
	p_bRequestToBring4 ACCESS ADR(bRequestToBring4);
	p_bRequestToGet4 ACCESS ADR(bRequestToGet4);
	p_bMag1SafetyBarRetCtrl ACCESS ADR (bMag1SafetyBarRetCtrl);
	p_bMag2SafetyBarRetCtrl ACCESS ADR (bMag2SafetyBarRetCtrl);
	p_bMag3SafetyBarRetCtrl ACCESS ADR (bMag3SafetyBarRetCtrl);
	p_bBypCurtainSen ACCESS ADR (bBypCurtainSen);
	p_bRstCurtainSen ACCESS ADR (bRstCurtainSen);
	p_bBypCurtainPBLED ACCESS ADR (bBypCurtainPBLED);
	p_bTrolleyExtCtrl ACCESS ADR (bTrolleyExtCtrl);
	p_bTrolleyExtCtrl2 ACCESS ADR (bTrolleyExtCtrl2);

END_ACTION
```
